LIN {X 0,Y 523.696,Z 765.358,A -85,B 0,C 180,E1 -4763.063,E2 -4763.063} C_VEL
LIN {X 0,Y 523.627,Z 770.61,A -85,B 0,C 180,E1 -4763.836,E2 -4763.836} C_VEL
LIN {X 0,Y 523.485,Z 774.989,A -85,B 0,C 180,E1 -4764.608,E2 -4764.608} C_VEL
LIN {X 0,Y 523.472,Z 780.149,A -85,B 0,C 180,E1 -4765.765,E2 -4765.765} C_VEL
LIN {X 0,Y 523.381,Z 783.938,A -85,B 0,C 180,E1 -4766.921,E2 -4766.921} C_VEL
LIN {X 0,Y 523.335,Z 785.68,A -85,B 0,C 180,E1 -4767.691,E2 -4767.691} C_VEL
LIN {X 0,Y 523.273,Z 786.929,A -85,B 0,C 180,E1 -4768.461,E2 -4768.461} C_VEL
LIN {X 0,Y 523.248,Z 787.706,A -85,B 0,C 180,E1 -4769.23,E2 -4769.23} C_VEL
LIN {X 0,Y 523.244,Z 788,A -85,B 0,C 180,E1 -4770,E2 -4770} C_VEL
LIN {X 0,Y 523.248,Z 787.707,A -85,B 0,C 180,E1 -4770.77,E2 -4770.77} C_VEL
LIN {X 0,Y 523.273,Z 786.93,A -85,B 0,C 180,E1 -4771.539,E2 -4771.539} C_VEL
LIN {X 0,Y 523.335,Z 785.682,A -85,B 0,C 180,E1 -4772.309,E2 -4772.309} C_VEL
LIN {X 0,Y 523.413,Z 782.788,A -85,B 0,C 180,E1 -4773.464,E2 -4773.464} C_VEL
LIN {X 0,Y 523.47,Z 780.149,A -85,B 0,C 180,E1 -4774.235,E2 -4774.235} C_VEL
LIN {X 0,Y 523.485,Z 774.99,A -85,B 0,C 180,E1 -4775.392,E2 -4775.392} C_VEL
LIN {X 0,Y 523.665,Z 768.76,A -85,B 0,C 180,E1 -4776.466,E2 -4776.466} C_VEL
LIN {X 0,Y 523.773,Z 760.74,A -85,B 0,C 180,E1 -4777.517,E2 -4777.517} C_VEL
LIN {X 0,Y 523.904,Z 753.36,A -85,B 0,C 180,E1 -4778.291,E2 -4778.291} C_VEL
LIN {X 0,Y 524.1,Z 745.417,A -85,B 0,C 180,E1 -4778.968,E2 -4778.968} C_VEL
LIN {X 0,Y 524.249,Z 736.974,A -85,B 0,C 180,E1 -4779.549,E2 -4779.549} C_VEL
LIN {X 0,Y 524.454,Z 726.202,A -85,B 0,C 180,E1 -4780.13,E2 -4780.13} C_VEL
LIN {X 0,Y 524.599,Z 714.549,A -85,B 0,C 180,E1 -4780.566,E2 -4780.566} C_VEL
LIN {X 0,Y 524.751,Z 704.885,A -85,B 0,C 180,E1 -4780.807,E2 -4780.807} C_VEL
LIN {X 0,Y 524.936,Z 646.273,A -85,B 0,C 180,E1 -4781.627,E2 -4781.627} C_VEL
LIN {X 0,Y 524.825,Z 633.309,A -85,B 0,C 180,E1 -4781.807,E2 -4781.807} C_VEL
LIN {X 0,Y 524.01,Z 625.533,A -85,B 0,C 180,E1 -4781.963,E2 -4781.963} C_VEL
LIN {X 0,Y 524.261,Z 604.559,A -85,B 0,C 180,E1 -4784.904,E2 -4784.904} C_VEL
LIN {X 0,Y 524.514,Z 583.003,A -85,B 0,C 180,E1 -4787.949,E2 -4787.949} C_VEL
LIN {X 0,Y 524.867,Z 561.889,A -85,B 0,C 180,E1 -4790.988,E2 -4790.988} C_VEL
LIN {X 0,Y 525.174,Z 542.146,A -85,B 0,C 180,E1 -4793.879,E2 -4793.879} C_VEL
LIN {X 0,Y 525.435,Z 522.421,A -85,B 0,C 180,E1 -4796.849,E2 -4796.849} C_VEL
LIN {X 0,Y 525.287,Z 516.932,A -85,B 0,C 180,E1 -4797.702,E2 -4797.702} C_VEL
LIN {X 0,Y 524.038,Z 510.273,A -85,B 0,C 180,E1 -4798.813,E2 -4798.813} C_VEL
LIN {X 0,Y 523.94,Z 510.034,A -85,B 0,C 180,E1 -4799.755,E2 -4799.755} C_VEL
LIN {X 0,Y 523.936,Z 510.033,A -85,B 0,C 180,E1 -4802.448,E2 -4802.448} C_VEL
LIN {X 0,Y 523.928,Z 510.036,A -85,B 0,C 180,E1 -4805.225,E2 -4805.225} C_VEL
LIN {X 0,Y 523.913,Z 510.033,A -85,B 0,C 180,E1 -4808.101,E2 -4808.101} C_VEL
LIN {X 0,Y 523.957,Z 510.03,A -85,B 0,C 180,E1 -4811.31,E2 -4811.31} C_VEL
LIN {X 0,Y 523.95,Z 510.033,A -85,B 0,C 180,E1 -4814.691,E2 -4814.691} C_VEL
LIN {X 0,Y 523.951,Z 510.025,A -85,B 0,C 180,E1 -4817.881,E2 -4817.881} C_VEL
LIN {X 0,Y 523.953,Z 510.033,A -85,B 0,C 180,E1 -4820.918,E2 -4820.918} C_VEL
LIN {X 0,Y 523.923,Z 510.029,A -85,B 0,C 180,E1 -4823.827,E2 -4823.827} C_VEL
LIN {X 0,Y 523.936,Z 510.034,A -85,B 0,C 180,E1 -4826.635,E2 -4826.635} C_VEL
LIN {X 0,Y 523.955,Z 510.029,A -85,B 0,C 180,E1 -4829.356,E2 -4829.356} C_VEL
LIN {X 0,Y 523.971,Z 510.026,A -85,B 0,C 180,E1 -4832.28,E2 -4832.28} C_VEL
LIN {X 0,Y 523.948,Z 510.03,A -85,B 0,C 180,E1 -4834.581,E2 -4834.581} C_VEL
LIN {X 0,Y 523.907,Z 510.039,A -85,B 0,C 180,E1 -4837.107,E2 -4837.107} C_VEL
LIN {X 0,Y 523.969,Z 510.024,A -85,B 0,C 180,E1 -4839.865,E2 -4839.865} C_VEL
LIN {X 0,Y 523.961,Z 510.033,A -85,B 0,C 180,E1 -4842.837,E2 -4842.837} C_VEL
LIN {X 0,Y 523.966,Z 510.03,A -85,B 0,C 180,E1 -4845.236,E2 -4845.236} C_VEL
LIN {X 0,Y 524.001,Z 510.024,A -85,B 0,C 180,E1 -4848.394,E2 -4848.394} C_VEL
LIN {X 0,Y 523.999,Z 510.023,A -85,B 0,C 180,E1 -4851.516,E2 -4851.516} C_VEL
LIN {X 0,Y 524.094,Z 510.016,A -85,B 0,C 180,E1 -4854.614,E2 -4854.614} C_VEL
LIN {X 0,Y 524.103,Z 510.01,A -85,B 0,C 180,E1 -4857.695,E2 -4857.695} C_VEL
LIN {X 0,Y 524.117,Z 510.015,A -85,B 0,C 180,E1 -4860.769,E2 -4860.769} C_VEL
LIN {X 0,Y 524.069,Z 510.019,A -85,B 0,C 180,E1 -4863.075,E2 -4863.075} C_VEL
LIN {X 0,Y 524.043,Z 510.022,A -85,B 0,C 180,E1 -4866.159,E2 -4866.159} C_VEL
LIN {X 0,Y 524.058,Z 510.143,A -85,B 0,C 180,E1 -4866.977,E2 -4866.977} C_VEL
LIN {X 0,Y 524.207,Z 511,A -85,B 0,C 180,E1 -4867.108,E2 -4867.108} C_VEL
LIN {X 0,Y 525.5,Z 515.641,A -85,B 0,C 180,E1 -4867.223,E2 -4867.223} C_VEL
LIN {X 0,Y 525.418,Z 540.428,A -85,B 0,C 180,E1 -4867.59,E2 -4867.59} C_VEL
LIN {X 0,Y 525.331,Z 553.745,A -85,B 0,C 180,E1 -4867.954,E2 -4867.954} C_VEL
LIN {X 0,Y 525.166,Z 566.276,A -85,B 0,C 180,E1 -4868.465,E2 -4868.465} C_VEL
LIN {X 0,Y 525.003,Z 577.002,A -85,B 0,C 180,E1 -4869.05,E2 -4869.05} C_VEL
LIN {X 0,Y 524.736,Z 588.282,A -85,B 0,C 180,E1 -4869.833,E2 -4869.833} C_VEL
LIN {X 0,Y 524.468,Z 598.441,A -85,B 0,C 180,E1 -4870.716,E2 -4870.716} C_VEL
LIN {X 0,Y 524.242,Z 607.233,A -85,B 0,C 180,E1 -4871.665,E2 -4871.665} C_VEL
LIN {X 0,Y 524.025,Z 615.656,A -85,B 0,C 180,E1 -4872.785,E2 -4872.785} C_VEL
LIN {X 0,Y 523.87,Z 622.807,A -85,B 0,C 180,E1 -4873.974,E2 -4873.974} C_VEL
LIN {X 0,Y 523.716,Z 628.632,A -85,B 0,C 180,E1 -4875.19,E2 -4875.19} C_VEL
LIN {X 0,Y 523.585,Z 633.022,A -85,B 0,C 180,E1 -4876.373,E2 -4876.373} C_VEL
LIN {X 0,Y 523.507,Z 636.422,A -85,B 0,C 180,E1 -4877.609,E2 -4877.609} C_VEL
LIN {X 0,Y 523.454,Z 638.654,A -85,B 0,C 180,E1 -4878.798,E2 -4878.798} C_VEL
LIN {X 0,Y 523.426,Z 639.92,A -85,B 0,C 180,E1 -4879.972,E2 -4879.972} C_VEL
LIN {X 0,Y 523.415,Z 640.261,A -85,B 0,C 180,E1 -4881.256,E2 -4881.256} C_VEL
LIN {X 0,Y 523.425,Z 639.894,A -85,B 0,C 180,E1 -4882.114,E2 -4882.114} C_VEL
LIN {X 0,Y 523.426,Z 639.12,A -85,B 0,C 180,E1 -4882.916,E2 -4882.916} C_VEL
LIN {X 0,Y 523.506,Z 637.178,A -85,B 0,C 180,E1 -4884.095,E2 -4884.095} C_VEL
LIN {X 0,Y 523.579,Z 633.768,A -85,B 0,C 180,E1 -4885.438,E2 -4885.438} C_VEL
LIN {X 0,Y 523.684,Z 629.24,A -85,B 0,C 180,E1 -4886.717,E2 -4886.717} C_VEL
LIN {X 0,Y 523.8,Z 623.233,A -85,B 0,C 180,E1 -4888.009,E2 -4888.009} C_VEL
LIN {X 0,Y 523.962,Z 616.769,A -85,B 0,C 180,E1 -4889.107,E2 -4889.107} C_VEL
LIN {X 0,Y 524.155,Z 608.949,A -85,B 0,C 180,E1 -4890.186,E2 -4890.186} C_VEL
LIN {X 0,Y 524.384,Z 600.525,A -85,B 0,C 180,E1 -4891.14,E2 -4891.14} C_VEL
LIN {X 0,Y 524.617,Z 590.534,A -85,B 0,C 180,E1 -4892.062,E2 -4892.062} C_VEL
LIN {X 0,Y 524.876,Z 580.07,A -85,B 0,C 180,E1 -4892.839,E2 -4892.839} C_VEL
LIN {X 0,Y 525.164,Z 568.003,A -85,B 0,C 180,E1 -4893.536,E2 -4893.536} C_VEL
LIN {X 0,Y 525.234,Z 562.226,A -85,B 0,C 180,E1 -4893.81,E2 -4893.81} C_VEL
LIN {X 0,Y 524.665,Z 556.768,A -85,B 0,C 180,E1 -4894.05,E2 -4894.05} C_VEL
LIN {X 0,Y 522.004,Z 547.838,A -85,B 0,C 180,E1 -4894.421,E2 -4894.421} C_VEL
LIN {X 0,Y 519.299,Z 538.713,A -85,B 0,C 180,E1 -4894.716,E2 -4894.716} C_VEL
LIN {X 0,Y 518.603,Z 532.955,A -85,B 0,C 180,E1 -4894.831,E2 -4894.831} C_VEL
LIN {X 0,Y 518.476,Z 516.07,A -85,B 0,C 180,E1 -4895.072,E2 -4895.072} C_VEL
LIN {X 0,Y 517.083,Z 511.785,A -85,B 0,C 180,E1 -4895.195,E2 -4895.195} C_VEL
LIN {X 0,Y 516.925,Z 510.992,A -85,B 0,C 180,E1 -4895.341,E2 -4895.341} C_VEL
LIN {X 0,Y 516.878,Z 510.912,A -85,B 0,C 180,E1 -4898.717,E2 -4898.717} C_VEL
LIN {X 0,Y 516.912,Z 510.907,A -85,B 0,C 180,E1 -4901.776,E2 -4901.776} C_VEL
LIN {X 0,Y 516.92,Z 510.906,A -85,B 0,C 180,E1 -4905.011,E2 -4905.011} C_VEL
LIN {X 0,Y 516.921,Z 510.902,A -85,B 0,C 180,E1 -4908.398,E2 -4908.398} C_VEL
LIN {X 0,Y 516.885,Z 510.914,A -85,B 0,C 180,E1 -4911.286,E2 -4911.286} C_VEL
LIN {X 0,Y 516.87,Z 510.909,A -85,B 0,C 180,E1 -4914.221,E2 -4914.221} C_VEL
LIN {X 0,Y 516.896,Z 510.908,A -85,B 0,C 180,E1 -4917.054,E2 -4917.054} C_VEL
LIN {X 0,Y 516.893,Z 510.91,A -85,B 0,C 180,E1 -4919.797,E2 -4919.797} C_VEL
LIN {X 0,Y 516.931,Z 510.901,A -85,B 0,C 180,E1 -4922.468,E2 -4922.468} C_VEL
LIN {X 0,Y 516.911,Z 510.906,A -85,B 0,C 180,E1 -4925.073,E2 -4925.073} C_VEL
LIN {X 0,Y 516.888,Z 510.906,A -85,B 0,C 180,E1 -4928.463,E2 -4928.463} C_VEL
LIN {X 0,Y 516.903,Z 510.905,A -85,B 0,C 180,E1 -4930.955,E2 -4930.955} C_VEL
LIN {X 0,Y 516.91,Z 510.91,A -85,B 0,C 180,E1 -4933.411,E2 -4933.411} C_VEL
LIN {X 0,Y 516.899,Z 510.911,A -85,B 0,C 180,E1 -4935.834,E2 -4935.834} C_VEL
LIN {X 0,Y 516.971,Z 510.897,A -85,B 0,C 180,E1 -4938.234,E2 -4938.234} C_VEL
LIN {X 0,Y 516.97,Z 510.901,A -85,B 0,C 180,E1 -4941.4,E2 -4941.4} C_VEL
LIN {X 0,Y 517.026,Z 510.889,A -85,B 0,C 180,E1 -4944.54,E2 -4944.54} C_VEL
LIN {X 0,Y 517.088,Z 510.89,A -85,B 0,C 180,E1 -4947.663,E2 -4947.663} C_VEL
LIN {X 0,Y 517.097,Z 510.88,A -85,B 0,C 180,E1 -4950.779,E2 -4950.779} C_VEL
LIN {X 0,Y 517.016,Z 510.891,A -85,B 0,C 180,E1 -4953.117,E2 -4953.117} C_VEL
LIN {X 0,Y 516.993,Z 510.896,A -85,B 0,C 180,E1 -4956.243,E2 -4956.243} C_VEL
LIN {X 0,Y 516.954,Z 510.901,A -85,B 0,C 180,E1 -4959.389,E2 -4959.389} C_VEL
LIN {X 0,Y 516.958,Z 510.907,A -85,B 0,C 180,E1 -4961.807,E2 -4961.807} C_VEL
LIN {X 0,Y 516.949,Z 510.899,A -85,B 0,C 180,E1 -4965.146,E2 -4965.146} C_VEL
LIN {X 0,Y 516.929,Z 510.905,A -85,B 0,C 180,E1 -4968.222,E2 -4968.222} C_VEL
LIN {X 0,Y 516.916,Z 510.903,A -85,B 0,C 180,E1 -4970.701,E2 -4970.701} C_VEL
LIN {X 0,Y 516.894,Z 510.913,A -85,B 0,C 180,E1 -4974.072,E2 -4974.072} C_VEL
LIN {X 0,Y 516.928,Z 510.902,A -85,B 0,C 180,E1 -4976.657,E2 -4976.657} C_VEL
LIN {X 0,Y 516.913,Z 510.906,A -85,B 0,C 180,E1 -4979.523,E2 -4979.523} C_VEL
LIN {X 0,Y 516.896,Z 510.907,A -85,B 0,C 180,E1 -4982.543,E2 -4982.543} C_VEL
LIN {X 0,Y 516.866,Z 510.91,A -85,B 0,C 180,E1 -4985.329,E2 -4985.329} C_VEL
LIN {X 0,Y 516.881,Z 510.915,A -85,B 0,C 180,E1 -4987.942,E2 -4987.942} C_VEL
LIN {X 0,Y 516.903,Z 510.905,A -85,B 0,C 180,E1 -4990.739,E2 -4990.739} C_VEL
LIN {X 0,Y 516.881,Z 510.913,A -85,B 0,C 180,E1 -4993.902,E2 -4993.902} C_VEL
LIN {X 0,Y 516.88,Z 510.917,A -85,B 0,C 180,E1 -4996.106,E2 -4996.106} C_VEL
LIN {X 0,Y 516.914,Z 510.908,A -85,B 0,C 180,E1 -4998.397,E2 -4998.397} C_VEL
LIN {X 0,Y 516.879,Z 510.907,A -85,B 0,C 180,E1 -5001.283,E2 -5001.283} C_VEL
LIN {X 0,Y 516.886,Z 510.916,A -85,B 0,C 180,E1 -5004.22,E2 -5004.22} C_VEL
LIN {X 0,Y 516.893,Z 510.906,A -85,B 0,C 180,E1 -5007.052,E2 -5007.052} C_VEL
LIN {X 0,Y 516.897,Z 510.908,A -85,B 0,C 180,E1 -5009.796,E2 -5009.796} C_VEL
LIN {X 0,Y 516.924,Z 510.908,A -85,B 0,C 180,E1 -5012.467,E2 -5012.467} C_VEL
LIN {X 0,Y 516.905,Z 510.904,A -85,B 0,C 180,E1 -5015.071,E2 -5015.071} C_VEL
LIN {X 0,Y 516.88,Z 510.914,A -85,B 0,C 180,E1 -5018.462,E2 -5018.462} C_VEL
LIN {X 0,Y 516.897,Z 510.906,A -85,B 0,C 180,E1 -5020.954,E2 -5020.954} C_VEL
LIN {X 0,Y 516.909,Z 510.903,A -85,B 0,C 180,E1 -5023.41,E2 -5023.41} C_VEL
LIN {X 0,Y 516.887,Z 510.908,A -85,B 0,C 180,E1 -5025.833,E2 -5025.833} C_VEL
LIN {X 0,Y 516.996,Z 510.9,A -85,B 0,C 180,E1 -5028.234,E2 -5028.234} C_VEL
LIN {X 0,Y 516.963,Z 510.897,A -85,B 0,C 180,E1 -5031.399,E2 -5031.399} C_VEL
LIN {X 0,Y 517.051,Z 510.894,A -85,B 0,C 180,E1 -5034.54,E2 -5034.54} C_VEL
LIN {X 0,Y 517.076,Z 510.883,A -85,B 0,C 180,E1 -5037.663,E2 -5037.663} C_VEL
LIN {X 0,Y 517.086,Z 510.886,A -85,B 0,C 180,E1 -5040.778,E2 -5040.778} C_VEL
LIN {X 0,Y 517.008,Z 510.893,A -85,B 0,C 180,E1 -5043.117,E2 -5043.117} C_VEL
LIN {X 0,Y 517.001,Z 510.897,A -85,B 0,C 180,E1 -5046.243,E2 -5046.243} C_VEL
LIN {X 0,Y 516.947,Z 510.899,A -85,B 0,C 180,E1 -5049.389,E2 -5049.389} C_VEL
LIN {X 0,Y 516.942,Z 510.9,A -85,B 0,C 180,E1 -5051.807,E2 -5051.807} C_VEL
LIN {X 0,Y 516.937,Z 510.902,A -85,B 0,C 180,E1 -5055.148,E2 -5055.148} C_VEL
LIN {X 0,Y 516.917,Z 510.906,A -85,B 0,C 180,E1 -5058.222,E2 -5058.222} C_VEL
LIN {X 0,Y 516.904,Z 510.913,A -85,B 0,C 180,E1 -5060.702,E2 -5060.702} C_VEL
LIN {X 0,Y 516.902,Z 510.906,A -85,B 0,C 180,E1 -5064.072,E2 -5064.072} C_VEL
LIN {X 0,Y 516.921,Z 510.911,A -85,B 0,C 180,E1 -5066.658,E2 -5066.658} C_VEL
LIN {X 0,Y 516.917,Z 510.903,A -85,B 0,C 180,E1 -5069.527,E2 -5069.527} C_VEL
LIN {X 0,Y 516.893,Z 510.912,A -85,B 0,C 180,E1 -5072.545,E2 -5072.545} C_VEL
LIN {X 0,Y 516.877,Z 510.909,A -85,B 0,C 180,E1 -5075.333,E2 -5075.333} C_VEL
LIN {X 0,Y 516.875,Z 510.908,A -85,B 0,C 180,E1 -5077.944,E2 -5077.944} C_VEL
LIN {X 0,Y 516.879,Z 510.916,A -85,B 0,C 180,E1 -5080.742,E2 -5080.742} C_VEL
LIN {X 0,Y 516.897,Z 510.915,A -85,B 0,C 180,E1 -5082.83,E2 -5082.83} C_VEL
LIN {X 0,Y 516.917,Z 510.91,A -85,B 0,C 180,E1 -5085.011,E2 -5085.011} C_VEL
LIN {X 0,Y 516.913,Z 510.906,A -85,B 0,C 180,E1 -5088.399,E2 -5088.399} C_VEL
LIN {X 0,Y 516.879,Z 510.911,A -85,B 0,C 180,E1 -5091.285,E2 -5091.285} C_VEL
LIN {X 0,Y 516.884,Z 510.909,A -85,B 0,C 180,E1 -5094.222,E2 -5094.222} C_VEL
LIN {X 0,Y 516.895,Z 510.914,A -85,B 0,C 180,E1 -5097.054,E2 -5097.054} C_VEL
LIN {X 0,Y 516.932,Z 511.029,A -85,B 0,C 180,E1 -5100.366,E2 -5100.366} C_VEL
LIN {X 0,Y 518.923,Z 520.98,A -85,B 0,C 180,E1 -5102.145,E2 -5102.145} C_VEL
LIN {X 0,Y 518.947,Z 529.197,A -85,B 0,C 180,E1 -5103.455,E2 -5103.455} C_VEL
LIN {X 0,Y 518.414,Z 548.211,A -85,B 0,C 180,E1 -5106.427,E2 -5106.427} C_VEL
LIN {X 0,Y 517.913,Z 567.608,A -85,B 0,C 180,E1 -5109.442,E2 -5109.442} C_VEL
LIN {X 0,Y 517.521,Z 584.748,A -85,B 0,C 180,E1 -5112.019,E2 -5112.019} C_VEL
LIN {X 0,Y 517.208,Z 606.759,A -85,B 0,C 180,E1 -5115.24,E2 -5115.24} C_VEL
LIN {X 0,Y 516.951,Z 624.671,A -85,B 0,C 180,E1 -5117.852,E2 -5117.852} C_VEL
LIN {X 0,Y 518.066,Z 636.508,A -85,B 0,C 180,E1 -5118.065,E2 -5118.065} C_VEL
LIN {X 0,Y 517.848,Z 703.106,A -85,B 0,C 180,E1 -5119.023,E2 -5119.023} C_VEL
LIN {X 0,Y 517.6,Z 713.015,A -85,B 0,C 180,E1 -5119.265,E2 -5119.265} C_VEL
LIN {X 0,Y 517.507,Z 724.237,A -85,B 0,C 180,E1 -5119.683,E2 -5119.683} C_VEL
LIN {X 0,Y 517.255,Z 734.516,A -85,B 0,C 180,E1 -5120.222,E2 -5120.222} C_VEL
LIN {X 0,Y 517.086,Z 744.454,A -85,B 0,C 180,E1 -5120.909,E2 -5120.909} C_VEL
LIN {X 0,Y 516.857,Z 752.427,A -85,B 0,C 180,E1 -5121.595,E2 -5121.595} C_VEL
LIN {X 0,Y 516.704,Z 759.897,A -85,B 0,C 180,E1 -5122.379,E2 -5122.379} C_VEL
LIN {X 0,Y 516.591,Z 766.92,A -85,B 0,C 180,E1 -5123.281,E2 -5123.281} C_VEL
LIN {X 0,Y 516.496,Z 773.47,A -85,B 0,C 180,E1 -5124.339,E2 -5124.339} C_VEL
LIN {X 0,Y 516.322,Z 778.169,A -85,B 0,C 180,E1 -5125.315,E2 -5125.315} C_VEL
LIN {X 0,Y 516.385,Z 781.242,A -85,B 0,C 180,E1 -5126.098,E2 -5126.098} C_VEL
LIN {X 0,Y 516.295,Z 783.609,A -85,B 0,C 180,E1 -5126.879,E2 -5126.879} C_VEL
LIN {X 0,Y 516.262,Z 785.398,A -85,B 0,C 180,E1 -5127.659,E2 -5127.659} C_VEL
LIN {X 0,Y 516.19,Z 786.673,A -85,B 0,C 180,E1 -5128.44,E2 -5128.44} C_VEL
LIN {X 0,Y 516.158,Z 787.467,A -85,B 0,C 180,E1 -5129.22,E2 -5129.22} C_VEL
LIN {X 0,Y 516.151,Z 787.768,A -85,B 0,C 180,E1 -5130,E2 -5130} C_VEL
LIN {X 0,Y 516.158,Z 787.469,A -85,B 0,C 180,E1 -5130.78,E2 -5130.78} C_VEL
LIN {X 0,Y 516.19,Z 786.674,A -85,B 0,C 180,E1 -5131.56,E2 -5131.56} C_VEL
LIN {X 0,Y 516.262,Z 785.398,A -85,B 0,C 180,E1 -5132.34,E2 -5132.34} C_VEL
LIN {X 0,Y 516.33,Z 782.429,A -85,B 0,C 180,E1 -5133.512,E2 -5133.512} C_VEL
LIN {X 0,Y 516.376,Z 779.716,A -85,B 0,C 180,E1 -5134.293,E2 -5134.293} C_VEL
LIN {X 0,Y 516.432,Z 774.416,A -85,B 0,C 180,E1 -5135.466,E2 -5135.466} C_VEL
LIN {X 0,Y 516.565,Z 768.545,A -85,B 0,C 180,E1 -5136.474,E2 -5136.474} C_VEL
LIN {X 0,Y 516.672,Z 761.524,A -85,B 0,C 180,E1 -5137.424,E2 -5137.424} C_VEL
LIN {X 0,Y 516.814,Z 753.324,A -85,B 0,C 180,E1 -5138.307,E2 -5138.307} C_VEL
LIN {X 0,Y 517.014,Z 745.516,A -85,B 0,C 180,E1 -5138.993,E2 -5138.993} C_VEL
LIN {X 0,Y 517.183,Z 737.327,A -85,B 0,C 180,E1 -5139.582,E2 -5139.582} C_VEL
LIN {X 0,Y 517.322,Z 728.859,A -85,B 0,C 180,E1 -5140.073,E2 -5140.073} C_VEL
LIN {X 0,Y 517.556,Z 719.044,A -85,B 0,C 180,E1 -5140.513,E2 -5140.513} C_VEL
LIN {X 0,Y 517.709,Z 707.406,A -85,B 0,C 180,E1 -5140.881,E2 -5140.881} C_VEL
LIN {X 0,Y 517.853,Z 689.806,A -85,B 0,C 180,E1 -5141.175,E2 -5141.175} C_VEL
LIN {X 0,Y 517.893,Z 634.084,A -85,B 0,C 180,E1 -5141.948,E2 -5141.948} C_VEL
LIN {X 0,Y 516.928,Z 624.065,A -85,B 0,C 180,E1 -5142.141,E2 -5142.141} C_VEL
LIN {X 0,Y 517.185,Z 605.597,A -85,B 0,C 180,E1 -5144.761,E2 -5144.761} C_VEL
LIN {X 0,Y 517.441,Z 583.365,A -85,B 0,C 180,E1 -5147.962,E2 -5147.962} C_VEL
LIN {X 0,Y 517.767,Z 563.429,A -85,B 0,C 180,E1 -5150.873,E2 -5150.873} C_VEL
LIN {X 0,Y 518.073,Z 545.172,A -85,B 0,C 180,E1 -5153.589,E2 -5153.589} C_VEL
LIN {X 0,Y 518.443,Z 525.628,A -85,B 0,C 180,E1 -5156.573,E2 -5156.573} C_VEL
LIN {X 0,Y 518.407,Z 518.846,A -85,B 0,C 180,E1 -5157.639,E2 -5157.639} C_VEL
LIN {X 0,Y 516.969,Z 511.076,A -85,B 0,C 180,E1 -5158.966,E2 -5158.966} C_VEL
LIN {X 0,Y 516.879,Z 510.91,A -85,B 0,C 180,E1 -5162.024,E2 -5162.024} C_VEL
LIN {X 0,Y 516.888,Z 510.915,A -85,B 0,C 180,E1 -5164.823,E2 -5164.823} C_VEL
LIN {X 0,Y 516.877,Z 510.909,A -85,B 0,C 180,E1 -5167.943,E2 -5167.943} C_VEL
LIN {X 0,Y 516.881,Z 510.914,A -85,B 0,C 180,E1 -5170.741,E2 -5170.741} C_VEL
LIN {X 0,Y 516.9,Z 510.912,A -85,B 0,C 180,E1 -5172.828,E2 -5172.828} C_VEL
LIN {X 0,Y 516.916,Z 510.91,A -85,B 0,C 180,E1 -5175.009,E2 -5175.009} C_VEL
LIN {X 0,Y 516.916,Z 510.903,A -85,B 0,C 180,E1 -5178.397,E2 -5178.397} C_VEL
LIN {X 0,Y 516.9,Z 510.909,A -85,B 0,C 180,E1 -5181.286,E2 -5181.286} C_VEL
LIN {X 0,Y 516.885,Z 510.907,A -85,B 0,C 180,E1 -5184.221,E2 -5184.221} C_VEL
LIN {X 0,Y 516.89,Z 510.912,A -85,B 0,C 180,E1 -5187.053,E2 -5187.053} C_VEL
LIN {X 0,Y 516.893,Z 510.906,A -85,B 0,C 180,E1 -5189.797,E2 -5189.797} C_VEL
LIN {X 0,Y 516.922,Z 510.906,A -85,B 0,C 180,E1 -5192.467,E2 -5192.467} C_VEL
LIN {X 0,Y 516.904,Z 510.912,A -85,B 0,C 180,E1 -5195.072,E2 -5195.072} C_VEL
LIN {X 0,Y 516.877,Z 510.912,A -85,B 0,C 180,E1 -5198.462,E2 -5198.462} C_VEL
LIN {X 0,Y 516.898,Z 510.914,A -85,B 0,C 180,E1 -5200.955,E2 -5200.955} C_VEL
LIN {X 0,Y 516.908,Z 510.907,A -85,B 0,C 180,E1 -5203.41,E2 -5203.41} C_VEL
LIN {X 0,Y 516.886,Z 510.908,A -85,B 0,C 180,E1 -5205.834,E2 -5205.834} C_VEL
LIN {X 0,Y 516.994,Z 510.896,A -85,B 0,C 180,E1 -5208.235,E2 -5208.235} C_VEL
LIN {X 0,Y 516.963,Z 510.901,A -85,B 0,C 180,E1 -5211.4,E2 -5211.4} C_VEL
LIN {X 0,Y 517.054,Z 510.892,A -85,B 0,C 180,E1 -5214.541,E2 -5214.541} C_VEL
LIN {X 0,Y 517.076,Z 510.885,A -85,B 0,C 180,E1 -5217.663,E2 -5217.663} C_VEL
LIN {X 0,Y 517.087,Z 510.891,A -85,B 0,C 180,E1 -5220.779,E2 -5220.779} C_VEL
LIN {X 0,Y 517.01,Z 510.898,A -85,B 0,C 180,E1 -5223.117,E2 -5223.117} C_VEL
LIN {X 0,Y 517.006,Z 510.899,A -85,B 0,C 180,E1 -5226.244,E2 -5226.244} C_VEL
LIN {X 0,Y 517.026,Z 511.162,A -85,B 0,C 180,E1 -5226.851,E2 -5226.851} C_VEL
LIN {X 0,Y 517.282,Z 512.234,A -85,B 0,C 180,E1 -5226.961,E2 -5226.961} C_VEL
LIN {X 0,Y 518.586,Z 517.279,A -85,B 0,C 180,E1 -5227.073,E2 -5227.073} C_VEL
LIN {X 0,Y 518.491,Z 541.4,A -85,B 0,C 180,E1 -5227.434,E2 -5227.434} C_VEL
LIN {X 0,Y 518.415,Z 554.495,A -85,B 0,C 180,E1 -5227.792,E2 -5227.792} C_VEL
LIN {X 0,Y 518.272,Z 566.108,A -85,B 0,C 180,E1 -5228.257,E2 -5228.257} C_VEL
LIN {X 0,Y 518.113,Z 577.551,A -85,B 0,C 180,E1 -5228.876,E2 -5228.876} C_VEL
LIN {X 0,Y 517.844,Z 588.947,A -85,B 0,C 180,E1 -5229.669,E2 -5229.669} C_VEL
LIN {X 0,Y 517.55,Z 599.194,A -85,B 0,C 180,E1 -5230.564,E2 -5230.564} C_VEL
LIN {X 0,Y 517.292,Z 608.336,A -85,B 0,C 180,E1 -5231.56,E2 -5231.56} C_VEL
LIN {X 0,Y 517.053,Z 617.197,A -85,B 0,C 180,E1 -5232.761,E2 -5232.761} C_VEL
LIN {X 0,Y 516.895,Z 624.271,A -85,B 0,C 180,E1 -5233.966,E2 -5233.966} C_VEL
LIN {X 0,Y 516.704,Z 630.546,A -85,B 0,C 180,E1 -5235.341,E2 -5235.341} C_VEL
LIN {X 0,Y 516.579,Z 634.913,A -85,B 0,C 180,E1 -5236.601,E2 -5236.601} C_VEL
LIN {X 0,Y 516.505,Z 637.81,A -85,B 0,C 180,E1 -5237.739,E2 -5237.739} C_VEL
LIN {X 0,Y 516.436,Z 640.064,A -85,B 0,C 180,E1 -5239.063,E2 -5239.063} C_VEL
LIN {X 0,Y 516.408,Z 641.014,A -85,B 0,C 180,E1 -5240.112,E2 -5240.112} C_VEL
LIN {X 0,Y 516.381,Z 641.197,A -85,B 0,C 180,E1 -5241.56,E2 -5241.56} C_VEL
LIN {X 0,Y 516.414,Z 640.678,A -85,B 0,C 180,E1 -5242.4,E2 -5242.4} C_VEL
LIN {X 0,Y 516.438,Z 639.688,A -85,B 0,C 180,E1 -5243.244,E2 -5243.244} C_VEL
LIN {X 0,Y 516.485,Z 637.892,A -85,B 0,C 180,E1 -5244.263,E2 -5244.263} C_VEL
LIN {X 0,Y 516.587,Z 633.766,A -85,B 0,C 180,E1 -5245.808,E2 -5245.808} C_VEL
LIN {X 0,Y 516.739,Z 628.884,A -85,B 0,C 180,E1 -5247.105,E2 -5247.105} C_VEL
LIN {X 0,Y 516.866,Z 622.439,A -85,B 0,C 180,E1 -5248.419,E2 -5248.419} C_VEL
LIN {X 0,Y 517.084,Z 615.358,A -85,B 0,C 180,E1 -5249.56,E2 -5249.56} C_VEL
LIN {X 0,Y 517.286,Z 607.222,A -85,B 0,C 180,E1 -5250.63,E2 -5250.63} C_VEL
LIN {X 0,Y 517.55,Z 597.771,A -85,B 0,C 180,E1 -5251.635,E2 -5251.635} C_VEL
LIN {X 0,Y 517.825,Z 587.493,A -85,B 0,C 180,E1 -5252.515,E2 -5252.515} C_VEL
LIN {X 0,Y 518.054,Z 577.412,A -85,B 0,C 180,E1 -5253.212,E2 -5253.212} C_VEL
LIN {X 0,Y 518.283,Z 565.658,A -85,B 0,C 180,E1 -5253.853,E2 -5253.853} C_VEL
LIN {X 0,Y 518.444,Z 552.926,A -85,B 0,C 180,E1 -5254.361,E2 -5254.361} C_VEL
LIN {X 0,Y 518.563,Z 539.177,A -85,B 0,C 180,E1 -5254.726,E2 -5254.726} C_VEL
LIN {X 0,Y 518.603,Z 532.955,A -85,B 0,C 180,E1 -5254.831,E2 -5254.831} C_VEL
LIN {X 0,Y 517.998,Z 529.111,A -85,B 0,C 180,E1 -5254.902,E2 -5254.902} C_VEL
LIN {X 0,Y 515.377,Z 523.171,A -85,B 0,C 180,E1 -5255.054,E2 -5255.054} C_VEL
LIN {X 0,Y 511.457,Z 516.232,A -85,B 0,C 180,E1 -5255.258,E2 -5255.258} C_VEL
LIN {X 0,Y 510.401,Z 513.803,A -85,B 0,C 180,E1 -5255.324,E2 -5255.324} C_VEL
LIN {X 0,Y 509.963,Z 512.303,A -85,B 0,C 180,E1 -5255.412,E2 -5255.412} C_VEL
LIN {X 0,Y 509.871,Z 511.819,A -85,B 0,C 180,E1 -5255.587,E2 -5255.587} C_VEL
LIN {X 0,Y 509.846,Z 511.787,A -85,B 0,C 180,E1 -5258.339,E2 -5258.339} C_VEL
LIN {X 0,Y 509.855,Z 511.792,A -85,B 0,C 180,E1 -5261.426,E2 -5261.426} C_VEL
LIN {X 0,Y 509.854,Z 511.783,A -85,B 0,C 180,E1 -5264.669,E2 -5264.669} C_VEL
LIN {X 0,Y 509.862,Z 511.782,A -85,B 0,C 180,E1 -5268.103,E2 -5268.103} C_VEL
LIN {X 0,Y 509.859,Z 511.782,A -85,B 0,C 180,E1 -5270.65,E2 -5270.65} C_VEL
LIN {X 0,Y 509.824,Z 511.792,A -85,B 0,C 180,E1 -5273.648,E2 -5273.648} C_VEL
LIN {X 0,Y 509.859,Z 511.782,A -85,B 0,C 180,E1 -5276.54,E2 -5276.54} C_VEL
LIN {X 0,Y 509.846,Z 511.79,A -85,B 0,C 180,E1 -5279.335,E2 -5279.335} C_VEL
LIN {X 0,Y 509.896,Z 511.779,A -85,B 0,C 180,E1 -5282.055,E2 -5282.055} C_VEL
LIN {X 0,Y 509.878,Z 511.78,A -85,B 0,C 180,E1 -5284.705,E2 -5284.705} C_VEL
LIN {X 0,Y 509.829,Z 511.793,A -85,B 0,C 180,E1 -5287.459,E2 -5287.459} C_VEL
LIN {X 0,Y 509.92,Z 511.779,A -85,B 0,C 180,E1 -5289.845,E2 -5289.845} C_VEL
LIN {X 0,Y 509.877,Z 511.783,A -85,B 0,C 180,E1 -5293.175,E2 -5293.175} C_VEL
LIN {X 0,Y 509.868,Z 511.79,A -85,B 0,C 180,E1 -5295.635,E2 -5295.635} C_VEL
LIN {X 0,Y 509.917,Z 511.775,A -85,B 0,C 180,E1 -5298.875,E2 -5298.875} C_VEL
LIN {X 0,Y 509.956,Z 511.773,A -85,B 0,C 180,E1 -5302.079,E2 -5302.079} C_VEL
LIN {X 0,Y 509.977,Z 511.767,A -85,B 0,C 180,E1 -5304.464,E2 -5304.464} C_VEL
LIN {X 0,Y 510.059,Z 511.765,A -85,B 0,C 180,E1 -5307.631,E2 -5307.631} C_VEL
LIN {X 0,Y 510.068,Z 511.756,A -85,B 0,C 180,E1 -5310.79,E2 -5310.79} C_VEL
LIN {X 0,Y 509.958,Z 511.771,A -85,B 0,C 180,E1 -5313.16,E2 -5313.16} C_VEL
LIN {X 0,Y 509.941,Z 511.773,A -85,B 0,C 180,E1 -5316.33,E2 -5316.33} C_VEL
LIN {X 0,Y 509.912,Z 511.775,A -85,B 0,C 180,E1 -5318.72,E2 -5318.72} C_VEL
LIN {X 0,Y 509.909,Z 511.783,A -85,B 0,C 180,E1 -5321.931,E2 -5321.931} C_VEL
LIN {X 0,Y 509.899,Z 511.778,A -85,B 0,C 180,E1 -5325.241,E2 -5325.241} C_VEL
LIN {X 0,Y 509.893,Z 511.785,A -85,B 0,C 180,E1 -5328,E2 -5328} C_VEL
LIN {X 0,Y 509.854,Z 511.782,A -85,B 0,C 180,E1 -5331.001,E2 -5331.001} C_VEL
LIN {X 0,Y 509.825,Z 511.79,A -85,B 0,C 180,E1 -5333.563,E2 -5333.563} C_VEL
LIN {X 0,Y 509.914,Z 511.778,A -85,B 0,C 180,E1 -5336.378,E2 -5336.378} C_VEL
LIN {X 0,Y 509.878,Z 511.779,A -85,B 0,C 180,E1 -5338.843,E2 -5338.843} C_VEL
LIN {X 0,Y 509.821,Z 511.79,A -85,B 0,C 180,E1 -5341.589,E2 -5341.589} C_VEL
LIN {X 0,Y 509.847,Z 511.787,A -85,B 0,C 180,E1 -5344.413,E2 -5344.413} C_VEL
LIN {X 0,Y 509.817,Z 511.788,A -85,B 0,C 180,E1 -5347.34,E2 -5347.34} C_VEL
LIN {X 0,Y 509.861,Z 511.786,A -85,B 0,C 180,E1 -5350.379,E2 -5350.379} C_VEL
LIN {X 0,Y 509.838,Z 511.784,A -85,B 0,C 180,E1 -5353.063,E2 -5353.063} C_VEL
LIN {X 0,Y 509.828,Z 511.79,A -85,B 0,C 180,E1 -5355.791,E2 -5355.791} C_VEL
LIN {X 0,Y 509.855,Z 511.785,A -85,B 0,C 180,E1 -5358.574,E2 -5358.574} C_VEL
LIN {X 0,Y 509.848,Z 511.787,A -85,B 0,C 180,E1 -5361.785,E2 -5361.785} C_VEL
LIN {X 0,Y 509.842,Z 511.787,A -85,B 0,C 180,E1 -5364.622,E2 -5364.622} C_VEL
LIN {X 0,Y 509.861,Z 511.782,A -85,B 0,C 180,E1 -5367.48,E2 -5367.48} C_VEL
LIN {X 0,Y 509.876,Z 511.789,A -85,B 0,C 180,E1 -5370.268,E2 -5370.268} C_VEL
LIN {X 0,Y 509.881,Z 511.78,A -85,B 0,C 180,E1 -5372.944,E2 -5372.944} C_VEL
LIN {X 0,Y 509.863,Z 511.782,A -85,B 0,C 180,E1 -5375.573,E2 -5375.573} C_VEL
LIN {X 0,Y 509.844,Z 511.784,A -85,B 0,C 180,E1 -5378.998,E2 -5378.998} C_VEL
LIN {X 0,Y 509.881,Z 511.783,A -85,B 0,C 180,E1 -5381.998,E2 -5381.998} C_VEL
LIN {X 0,Y 509.902,Z 511.779,A -85,B 0,C 180,E1 -5384.818,E2 -5384.818} C_VEL
LIN {X 0,Y 509.935,Z 511.777,A -85,B 0,C 180,E1 -5388.1,E2 -5388.1} C_VEL
LIN {X 0,Y 509.91,Z 511.775,A -85,B 0,C 180,E1 -5391.279,E2 -5391.279} C_VEL
LIN {X 0,Y 509.97,Z 511.768,A -85,B 0,C 180,E1 -5393.67,E2 -5393.67} C_VEL
LIN {X 0,Y 509.95,Z 511.774,A -85,B 0,C 180,E1 -5396.84,E2 -5396.84} C_VEL
LIN {X 0,Y 510.056,Z 511.758,A -85,B 0,C 180,E1 -5399.21,E2 -5399.21} C_VEL
LIN {X 0,Y 510.046,Z 511.766,A -85,B 0,C 180,E1 -5402.369,E2 -5402.369} C_VEL
LIN {X 0,Y 509.969,Z 511.774,A -85,B 0,C 180,E1 -5406.329,E2 -5406.329} C_VEL
LIN {X 0,Y 509.909,Z 511.782,A -85,B 0,C 180,E1 -5408.72,E2 -5408.72} C_VEL
LIN {X 0,Y 509.894,Z 511.778,A -85,B 0,C 180,E1 -5411.932,E2 -5411.932} C_VEL
LIN {X 0,Y 509.884,Z 511.78,A -85,B 0,C 180,E1 -5415.242,E2 -5415.242} C_VEL
LIN {X 0,Y 509.879,Z 511.78,A -85,B 0,C 180,E1 -5418.001,E2 -5418.001} C_VEL
LIN {X 0,Y 509.842,Z 511.788,A -85,B 0,C 180,E1 -5421.002,E2 -5421.002} C_VEL
LIN {X 0,Y 509.828,Z 511.786,A -85,B 0,C 180,E1 -5423.563,E2 -5423.563} C_VEL
LIN {X 0,Y 509.905,Z 511.78,A -85,B 0,C 180,E1 -5426.379,E2 -5426.379} C_VEL
LIN {X 0,Y 509.878,Z 511.787,A -85,B 0,C 180,E1 -5428.844,E2 -5428.844} C_VEL
LIN {X 0,Y 509.818,Z 511.787,A -85,B 0,C 180,E1 -5431.59,E2 -5431.59} C_VEL
LIN {X 0,Y 509.848,Z 511.787,A -85,B 0,C 180,E1 -5434.414,E2 -5434.414} C_VEL
LIN {X 0,Y 509.812,Z 511.789,A -85,B 0,C 180,E1 -5437.341,E2 -5437.341} C_VEL
LIN {X 0,Y 509.832,Z 511.788,A -85,B 0,C 180,E1 -5440.383,E2 -5440.383} C_VEL
LIN {X 0,Y 509.832,Z 511.791,A -85,B 0,C 180,E1 -5443.065,E2 -5443.065} C_VEL
LIN {X 0,Y 509.825,Z 511.786,A -85,B 0,C 180,E1 -5445.793,E2 -5445.793} C_VEL
LIN {X 0,Y 509.854,Z 511.787,A -85,B 0,C 180,E1 -5448.575,E2 -5448.575} C_VEL
LIN {X 0,Y 509.848,Z 511.783,A -85,B 0,C 180,E1 -5451.787,E2 -5451.787} C_VEL
LIN {X 0,Y 509.839,Z 511.79,A -85,B 0,C 180,E1 -5454.624,E2 -5454.624} C_VEL
LIN {X 0,Y 509.863,Z 511.788,A -85,B 0,C 180,E1 -5457.482,E2 -5457.482} C_VEL
LIN {X 0,Y 509.912,Z 511.99,A -85,B 0,C 180,E1 -5460.196,E2 -5460.196} C_VEL
LIN {X 0,Y 512.075,Z 523.14,A -85,B 0,C 180,E1 -5462.185,E2 -5462.185} C_VEL
LIN {X 0,Y 511.878,Z 533.986,A -85,B 0,C 180,E1 -5463.938,E2 -5463.938} C_VEL
LIN {X 0,Y 511.351,Z 552.4,A -85,B 0,C 180,E1 -5466.869,E2 -5466.869} C_VEL
LIN {X 0,Y 510.773,Z 572.895,A -85,B 0,C 180,E1 -5470.09,E2 -5470.09} C_VEL
LIN {X 0,Y 510.437,Z 589.341,A -85,B 0,C 180,E1 -5472.575,E2 -5472.575} C_VEL
LIN {X 0,Y 510.096,Z 610.033,A -85,B 0,C 180,E1 -5475.641,E2 -5475.641} C_VEL
LIN {X 0,Y 509.882,Z 623.464,A -85,B 0,C 180,E1 -5477.654,E2 -5477.654} C_VEL
LIN {X 0,Y 510.954,Z 634.279,A -85,B 0,C 180,E1 -5477.86,E2 -5477.86} C_VEL
LIN {X 0,Y 510.979,Z 665.653,A -85,B 0,C 180,E1 -5478.32,E2 -5478.32} C_VEL
LIN {X 0,Y 510.831,Z 703.726,A -85,B 0,C 180,E1 -5478.895,E2 -5478.895} C_VEL
LIN {X 0,Y 510.598,Z 716.003,A -85,B 0,C 180,E1 -5479.241,E2 -5479.241} C_VEL
LIN {X 0,Y 510.38,Z 726.331,A -85,B 0,C 180,E1 -5479.688,E2 -5479.688} C_VEL
LIN {X 0,Y 510.179,Z 735.081,A -85,B 0,C 180,E1 -5480.185,E2 -5480.185} C_VEL
LIN {X 0,Y 510.001,Z 744.733,A -85,B 0,C 180,E1 -5480.882,E2 -5480.882} C_VEL
LIN {X 0,Y 509.725,Z 753.52,A -85,B 0,C 180,E1 -5481.676,E2 -5481.676} C_VEL
LIN {X 0,Y 509.562,Z 762.185,A -85,B 0,C 180,E1 -5482.67,E2 -5482.67} C_VEL
LIN {X 0,Y 509.457,Z 769,A -85,B 0,C 180,E1 -5483.664,E2 -5483.664} C_VEL
LIN {X 0,Y 509.382,Z 773.479,A -85,B 0,C 180,E1 -5484.458,E2 -5484.458} C_VEL
LIN {X 0,Y 509.304,Z 778.763,A -85,B 0,C 180,E1 -5485.647,E2 -5485.647} C_VEL
LIN {X 0,Y 509.279,Z 781.469,A -85,B 0,C 180,E1 -5486.44,E2 -5486.44} C_VEL
LIN {X 0,Y 509.214,Z 784.431,A -85,B 0,C 180,E1 -5487.627,E2 -5487.627} C_VEL
LIN {X 0,Y 509.152,Z 785.703,A -85,B 0,C 180,E1 -5488.418,E2 -5488.418} C_VEL
LIN {X 0,Y 509.123,Z 786.493,A -85,B 0,C 180,E1 -5489.209,E2 -5489.209} C_VEL
LIN {X 0,Y 509.142,Z 786.782,A -85,B 0,C 180,E1 -5490,E2 -5490} C_VEL
LIN {X 0,Y 509.124,Z 786.485,A -85,B 0,C 180,E1 -5490.791,E2 -5490.791} C_VEL
LIN {X 0,Y 509.155,Z 785.679,A -85,B 0,C 180,E1 -5491.582,E2 -5491.582} C_VEL
LIN {X 0,Y 509.22,Z 784.389,A -85,B 0,C 180,E1 -5492.373,E2 -5492.373} C_VEL
LIN {X 0,Y 509.288,Z 781.404,A -85,B 0,C 180,E1 -5493.56,E2 -5493.56} C_VEL
LIN {X 0,Y 509.303,Z 778.67,A -85,B 0,C 180,E1 -5494.353,E2 -5494.353} C_VEL
LIN {X 0,Y 509.389,Z 773.357,A -85,B 0,C 180,E1 -5495.542,E2 -5495.542} C_VEL
LIN {X 0,Y 509.505,Z 766.476,A -85,B 0,C 180,E1 -5496.71,E2 -5496.71} C_VEL
LIN {X 0,Y 509.628,Z 758.676,A -85,B 0,C 180,E1 -5497.727,E2 -5497.727} C_VEL
LIN {X 0,Y 509.765,Z 751.145,A -85,B 0,C 180,E1 -5498.523,E2 -5498.523} C_VEL
LIN {X 0,Y 510.037,Z 741.867,A -85,B 0,C 180,E1 -5499.317,E2 -5499.317} C_VEL
LIN {X 0,Y 510.254,Z 731.411,A -85,B 0,C 180,E1 -5500.014,E2 -5500.014} C_VEL
LIN {X 0,Y 510.48,Z 720.308,A -85,B 0,C 180,E1 -5500.56,E2 -5500.56} C_VEL
LIN {X 0,Y 510.646,Z 709.749,A -85,B 0,C 180,E1 -5500.933,E2 -5500.933} C_VEL
LIN {X 0,Y 510.874,Z 698.835,A -85,B 0,C 180,E1 -5501.179,E2 -5501.179} C_VEL
LIN {X 0,Y 510.929,Z 634.519,A -85,B 0,C 180,E1 -5502.101,E2 -5502.101} C_VEL
LIN {X 0,Y 509.845,Z 622.828,A -85,B 0,C 180,E1 -5502.312,E2 -5502.312} C_VEL
LIN {X 0,Y 509.851,Z 620.84,A -85,B 0,C 180,E1 -5502.539,E2 -5502.539} C_VEL
LIN {X 0,Y 510.083,Z 602.756,A -85,B 0,C 180,E1 -5505.176,E2 -5505.176} C_VEL
LIN {X 0,Y 510.369,Z 584.186,A -85,B 0,C 180,E1 -5507.9,E2 -5507.9} C_VEL
LIN {X 0,Y 510.723,Z 563.575,A -85,B 0,C 180,E1 -5510.963,E2 -5510.963} C_VEL
LIN {X 0,Y 511.076,Z 543.992,A -85,B 0,C 180,E1 -5513.932,E2 -5513.932} C_VEL
LIN {X 0,Y 511.444,Z 524.57,A -85,B 0,C 180,E1 -5516.966,E2 -5516.966} C_VEL
LIN {X 0,Y 511.243,Z 519.028,A -85,B 0,C 180,E1 -5517.864,E2 -5517.864} C_VEL
LIN {X 0,Y 509.908,Z 511.903,A -85,B 0,C 180,E1 -5519.124,E2 -5519.124} C_VEL
LIN {X 0,Y 509.862,Z 511.787,A -85,B 0,C 180,E1 -5522.518,E2 -5522.518} C_VEL
LIN {X 0,Y 509.835,Z 511.788,A -85,B 0,C 180,E1 -5525.58,E2 -5525.58} C_VEL
LIN {X 0,Y 509.847,Z 511.786,A -85,B 0,C 180,E1 -5528.337,E2 -5528.337} C_VEL
LIN {X 0,Y 509.853,Z 511.786,A -85,B 0,C 180,E1 -5531.424,E2 -5531.424} C_VEL
LIN {X 0,Y 509.85,Z 511.789,A -85,B 0,C 180,E1 -5534.667,E2 -5534.667} C_VEL
LIN {X 0,Y 509.857,Z 511.781,A -85,B 0,C 180,E1 -5538.102,E2 -5538.102} C_VEL
LIN {X 0,Y 509.87,Z 511.786,A -85,B 0,C 180,E1 -5540.65,E2 -5540.65} C_VEL
LIN {X 0,Y 509.829,Z 511.785,A -85,B 0,C 180,E1 -5543.647,E2 -5543.647} C_VEL
LIN {X 0,Y 509.856,Z 511.787,A -85,B 0,C 180,E1 -5546.539,E2 -5546.539} C_VEL
LIN {X 0,Y 509.842,Z 511.787,A -85,B 0,C 180,E1 -5549.334,E2 -5549.334} C_VEL
LIN {X 0,Y 509.887,Z 511.78,A -85,B 0,C 180,E1 -5552.054,E2 -5552.054} C_VEL
LIN {X 0,Y 509.87,Z 511.785,A -85,B 0,C 180,E1 -5554.704,E2 -5554.704} C_VEL
LIN {X 0,Y 509.846,Z 511.786,A -85,B 0,C 180,E1 -5557.449,E2 -5557.449} C_VEL
LIN {X 0,Y 509.907,Z 511.776,A -85,B 0,C 180,E1 -5559.845,E2 -5559.845} C_VEL
LIN {X 0,Y 509.878,Z 511.786,A -85,B 0,C 180,E1 -5563.175,E2 -5563.175} C_VEL
LIN {X 0,Y 509.854,Z 511.784,A -85,B 0,C 180,E1 -5565.634,E2 -5565.634} C_VEL
LIN {X 0,Y 509.916,Z 511.783,A -85,B 0,C 180,E1 -5568.875,E2 -5568.875} C_VEL
LIN {X 0,Y 509.942,Z 511.774,A -85,B 0,C 180,E1 -5572.079,E2 -5572.079} C_VEL
LIN {X 0,Y 510.001,Z 511.77,A -85,B 0,C 180,E1 -5574.465,E2 -5574.465} C_VEL
LIN {X 0,Y 510.047,Z 511.761,A -85,B 0,C 180,E1 -5577.631,E2 -5577.631} C_VEL
LIN {X 0,Y 510.057,Z 511.767,A -85,B 0,C 180,E1 -5580.79,E2 -5580.79} C_VEL
LIN {X 0,Y 509.952,Z 511.777,A -85,B 0,C 180,E1 -5583.16,E2 -5583.16} C_VEL
LIN {X 0,Y 509.968,Z 511.777,A -85,B 0,C 180,E1 -5586.33,E2 -5586.33} C_VEL
LIN {X 0,Y 509.978,Z 512.099,A -85,B 0,C 180,E1 -5586.694,E2 -5586.694} C_VEL
LIN {X 0,Y 510.296,Z 513.352,A -85,B 0,C 180,E1 -5586.799,E2 -5586.799} C_VEL
LIN {X 0,Y 511.659,Z 517.922,A -85,B 0,C 180,E1 -5586.905,E2 -5586.905} C_VEL
LIN {X 0,Y 511.58,Z 541.849,A -85,B 0,C 180,E1 -5587.261,E2 -5587.261} C_VEL
LIN {X 0,Y 511.52,Z 555.304,A -85,B 0,C 180,E1 -5587.628,E2 -5587.628} C_VEL
LIN {X 0,Y 511.392,Z 567.054,A -85,B 0,C 180,E1 -5588.102,E2 -5588.102} C_VEL
LIN {X 0,Y 511.213,Z 578.089,A -85,B 0,C 180,E1 -5588.698,E2 -5588.698} C_VEL
LIN {X 0,Y 510.951,Z 589.584,A -85,B 0,C 180,E1 -5589.501,E2 -5589.501} C_VEL
LIN {X 0,Y 510.624,Z 599.934,A -85,B 0,C 180,E1 -5590.408,E2 -5590.408} C_VEL
LIN {X 0,Y 510.384,Z 608.333,A -85,B 0,C 180,E1 -5591.316,E2 -5591.316} C_VEL
LIN {X 0,Y 510.146,Z 617.372,A -85,B 0,C 180,E1 -5592.532,E2 -5592.532} C_VEL
LIN {X 0,Y 509.928,Z 624.646,A -85,B 0,C 180,E1 -5593.754,E2 -5593.754} C_VEL
LIN {X 0,Y 509.767,Z 629.541,A -85,B 0,C 180,E1 -5594.777,E2 -5594.777} C_VEL
LIN {X 0,Y 509.626,Z 634.261,A -85,B 0,C 180,E1 -5596.011,E2 -5596.011} C_VEL
LIN {X 0,Y 509.539,Z 637.824,A -85,B 0,C 180,E1 -5597.251,E2 -5597.251} C_VEL
LIN {X 0,Y 509.451,Z 640.326,A -85,B 0,C 180,E1 -5598.499,E2 -5598.499} C_VEL
LIN {X 0,Y 509.415,Z 641.411,A -85,B 0,C 180,E1 -5599.336,E2 -5599.336} C_VEL
LIN {X 0,Y 509.38,Z 642.108,A -85,B 0,C 180,E1 -5600.251,E2 -5600.251} C_VEL
LIN {X 0,Y 509.374,Z 642.304,A -85,B 0,C 180,E1 -5601.023,E2 -5601.023} C_VEL
LIN {X 0,Y 509.386,Z 641.666,A -85,B 0,C 180,E1 -5602.426,E2 -5602.426} C_VEL
LIN {X 0,Y 509.441,Z 640.223,A -85,B 0,C 180,E1 -5603.583,E2 -5603.583} C_VEL
LIN {X 0,Y 509.542,Z 637.551,A -85,B 0,C 180,E1 -5604.878,E2 -5604.878} C_VEL
LIN {X 0,Y 509.651,Z 633.185,A -85,B 0,C 180,E1 -5606.322,E2 -5606.322} C_VEL
LIN {X 0,Y 509.773,Z 627.409,A -85,B 0,C 180,E1 -5607.73,E2 -5607.73} C_VEL
LIN {X 0,Y 509.98,Z 620.198,A -85,B 0,C 180,E1 -5609.064,E2 -5609.064} C_VEL
LIN {X 0,Y 510.22,Z 612.635,A -85,B 0,C 180,E1 -5610.183,E2 -5610.183} C_VEL
LIN {X 0,Y 510.517,Z 603.188,A -85,B 0,C 180,E1 -5611.311,E2 -5611.311} C_VEL
LIN {X 0,Y 510.78,Z 592.395,A -85,B 0,C 180,E1 -5612.337,E2 -5612.337} C_VEL
LIN {X 0,Y 511.068,Z 582.093,A -85,B 0,C 180,E1 -5613.12,E2 -5613.12} C_VEL
LIN {X 0,Y 511.33,Z 570.263,A -85,B 0,C 180,E1 -5613.825,E2 -5613.825} C_VEL
LIN {X 0,Y 511.52,Z 557.817,A -85,B 0,C 180,E1 -5614.382,E2 -5614.382} C_VEL
LIN {X 0,Y 511.635,Z 544.878,A -85,B 0,C 180,E1 -5614.787,E2 -5614.787} C_VEL
LIN {X 0,Y 511.689,Z 529.452,A -85,B 0,C 180,E1 -5615.063,E2 -5615.063} C_VEL
LIN {X 0,Y 511.669,Z 517.77,A -85,B 0,C 180,E1 -5615.23,E2 -5615.23} C_VEL
LIN {X 0,Y 510.401,Z 513.803,A -85,B 0,C 180,E1 -5615.324,E2 -5615.324} C_VEL
LIN {X 0,Y 509.62,Z 512.589,A -85,B 0,C 180,E1 -5615.443,E2 -5615.443} C_VEL
LIN {X 0,Y 508.356,Z 512.057,A -85,B 0,C 180,E1 -5615.712,E2 -5615.712} C_VEL
LIN {X 0,Y 505.264,Z 512.362,A -85,B 0,C 180,E1 -5616.711,E2 -5616.711} C_VEL
LIN {X 0,Y 503.83,Z 512.853,A -85,B 0,C 180,E1 -5617.474,E2 -5617.474} C_VEL
LIN {X 0,Y 502.964,Z 512.745,A -85,B 0,C 180,E1 -5618.255,E2 -5618.255} C_VEL
LIN {X 0,Y 502.791,Z 512.668,A -85,B 0,C 180,E1 -5618.779,E2 -5618.779} C_VEL
LIN {X 0,Y 502.826,Z 512.66,A -85,B 0,C 180,E1 -5622.137,E2 -5622.137} C_VEL
LIN {X 0,Y 502.798,Z 512.669,A -85,B 0,C 180,E1 -5625.469,E2 -5625.469} C_VEL
LIN {X 0,Y 502.828,Z 512.66,A -85,B 0,C 180,E1 -5627.865,E2 -5627.865} C_VEL
LIN {X 0,Y 502.809,Z 512.664,A -85,B 0,C 180,E1 -5631.026,E2 -5631.026} C_VEL
LIN {X 0,Y 502.774,Z 512.665,A -85,B 0,C 180,E1 -5634.17,E2 -5634.17} C_VEL
LIN {X 0,Y 502.833,Z 512.66,A -85,B 0,C 180,E1 -5636.994,E2 -5636.994} C_VEL
LIN {X 0,Y 502.816,Z 512.661,A -85,B 0,C 180,E1 -5640.066,E2 -5640.066} C_VEL
LIN {X 0,Y 502.836,Z 512.656,A -85,B 0,C 180,E1 -5642.534,E2 -5642.534} C_VEL
LIN {X 0,Y 502.829,Z 512.663,A -85,B 0,C 180,E1 -5645.3,E2 -5645.3} C_VEL
LIN {X 0,Y 502.783,Z 512.668,A -85,B 0,C 180,E1 -5647.827,E2 -5647.827} C_VEL
LIN {X 0,Y 502.827,Z 512.658,A -85,B 0,C 180,E1 -5650.401,E2 -5650.401} C_VEL
LIN {X 0,Y 502.822,Z 512.659,A -85,B 0,C 180,E1 -5652.932,E2 -5652.932} C_VEL
LIN {X 0,Y 502.849,Z 512.661,A -85,B 0,C 180,E1 -5655.43,E2 -5655.43} C_VEL
LIN {X 0,Y 502.882,Z 512.651,A -85,B 0,C 180,E1 -5658.717,E2 -5658.717} C_VEL
LIN {X 0,Y 502.906,Z 512.653,A -85,B 0,C 180,E1 -5661.967,E2 -5661.967} C_VEL
LIN {X 0,Y 502.93,Z 512.646,A -85,B 0,C 180,E1 -5664.387,E2 -5664.387} C_VEL
LIN {X 0,Y 503.029,Z 512.64,A -85,B 0,C 180,E1 -5667.598,E2 -5667.598} C_VEL
LIN {X 0,Y 503.033,Z 512.637,A -85,B 0,C 180,E1 -5670,E2 -5670} C_VEL
LIN {X 0,Y 503.029,Z 512.634,A -85,B 0,C 180,E1 -5672.402,E2 -5672.402} C_VEL
LIN {X 0,Y 502.931,Z 512.651,A -85,B 0,C 180,E1 -5675.613,E2 -5675.613} C_VEL
LIN {X 0,Y 502.872,Z 512.652,A -85,B 0,C 180,E1 -5678.843,E2 -5678.843} C_VEL
LIN {X 0,Y 502.851,Z 512.66,A -85,B 0,C 180,E1 -5682.101,E2 -5682.101} C_VEL
LIN {X 0,Y 502.853,Z 512.657,A -85,B 0,C 180,E1 -5685.399,E2 -5685.399} C_VEL
LIN {X 0,Y 502.85,Z 512.66,A -85,B 0,C 180,E1 -5688.122,E2 -5688.122} C_VEL
LIN {X 0,Y 502.832,Z 512.658,A -85,B 0,C 180,E1 -5690.536,E2 -5690.536} C_VEL
LIN {X 0,Y 502.791,Z 512.662,A -85,B 0,C 180,E1 -5693.04,E2 -5693.04} C_VEL
LIN {X 0,Y 502.824,Z 512.663,A -85,B 0,C 180,E1 -5695.676,E2 -5695.676} C_VEL
LIN {X 0,Y 502.842,Z 512.659,A -85,B 0,C 180,E1 -5698.372,E2 -5698.372} C_VEL
LIN {X 0,Y 502.794,Z 512.664,A -85,B 0,C 180,E1 -5701.498,E2 -5701.498} C_VEL
LIN {X 0,Y 502.804,Z 512.67,A -85,B 0,C 180,E1 -5703.993,E2 -5703.993} C_VEL
LIN {X 0,Y 502.777,Z 512.664,A -85,B 0,C 180,E1 -5707.177,E2 -5707.177} C_VEL
LIN {X 0,Y 502.821,Z 512.667,A -85,B 0,C 180,E1 -5710.011,E2 -5710.011} C_VEL
LIN {X 0,Y 502.822,Z 512.666,A -85,B 0,C 180,E1 -5712.201,E2 -5712.201} C_VEL
LIN {X 0,Y 502.798,Z 512.662,A -85,B 0,C 180,E1 -5715.467,E2 -5715.467} C_VEL
LIN {X 0,Y 502.817,Z 512.659,A -85,B 0,C 180,E1 -5718.933,E2 -5718.933} C_VEL
LIN {X 0,Y 502.79,Z 512.67,A -85,B 0,C 180,E1 -5722.045,E2 -5722.045} C_VEL
LIN {X 0,Y 502.805,Z 512.661,A -85,B 0,C 180,E1 -5725.034,E2 -5725.034} C_VEL
LIN {X 0,Y 502.783,Z 512.668,A -85,B 0,C 180,E1 -5727.915,E2 -5727.915} C_VEL
LIN {X 0,Y 502.834,Z 512.66,A -85,B 0,C 180,E1 -5730.712,E2 -5730.712} C_VEL
LIN {X 0,Y 502.875,Z 512.652,A -85,B 0,C 180,E1 -5733.434,E2 -5733.434} C_VEL
LIN {X 0,Y 502.785,Z 512.669,A -85,B 0,C 180,E1 -5736.086,E2 -5736.086} C_VEL
LIN {X 0,Y 502.777,Z 512.668,A -85,B 0,C 180,E1 -5738.688,E2 -5738.688} C_VEL
LIN {X 0,Y 502.823,Z 512.658,A -85,B 0,C 180,E1 -5741.248,E2 -5741.248} C_VEL
LIN {X 0,Y 502.816,Z 512.661,A -85,B 0,C 180,E1 -5743.767,E2 -5743.767} C_VEL
LIN {X 0,Y 502.823,Z 512.666,A -85,B 0,C 180,E1 -5746.254,E2 -5746.254} C_VEL
LIN {X 0,Y 502.884,Z 512.655,A -85,B 0,C 180,E1 -5748.717,E2 -5748.717} C_VEL
LIN {X 0,Y 502.894,Z 512.652,A -85,B 0,C 180,E1 -5751.966,E2 -5751.966} C_VEL
LIN {X 0,Y 502.95,Z 512.651,A -85,B 0,C 180,E1 -5754.386,E2 -5754.386} C_VEL
LIN {X 0,Y 503.016,Z 512.634,A -85,B 0,C 180,E1 -5757.597,E2 -5757.597} C_VEL
LIN {X 0,Y 503.017,Z 512.636,A -85,B 0,C 180,E1 -5760,E2 -5760} C_VEL
LIN {X 0,Y 503.016,Z 512.642,A -85,B 0,C 180,E1 -5762.402,E2 -5762.402} C_VEL
LIN {X 0,Y 502.93,Z 512.645,A -85,B 0,C 180,E1 -5765.613,E2 -5765.613} C_VEL
LIN {X 0,Y 502.893,Z 512.652,A -85,B 0,C 180,E1 -5768.033,E2 -5768.033} C_VEL
LIN {X 0,Y 502.868,Z 512.653,A -85,B 0,C 180,E1 -5771.283,E2 -5771.283} C_VEL
LIN {X 0,Y 502.842,Z 512.665,A -85,B 0,C 180,E1 -5774.571,E2 -5774.571} C_VEL
LIN {X 0,Y 502.853,Z 512.655,A -85,B 0,C 180,E1 -5777.907,E2 -5777.907} C_VEL
LIN {X 0,Y 502.82,Z 512.666,A -85,B 0,C 180,E1 -5780.536,E2 -5780.536} C_VEL
LIN {X 0,Y 502.788,Z 512.666,A -85,B 0,C 180,E1 -5783.041,E2 -5783.041} C_VEL
LIN {X 0,Y 502.833,Z 512.657,A -85,B 0,C 180,E1 -5785.676,E2 -5785.676} C_VEL
LIN {X 0,Y 502.834,Z 512.661,A -85,B 0,C 180,E1 -5788.373,E2 -5788.373} C_VEL
LIN {X 0,Y 502.789,Z 512.663,A -85,B 0,C 180,E1 -5791.5,E2 -5791.5} C_VEL
LIN {X 0,Y 502.8,Z 512.665,A -85,B 0,C 180,E1 -5794.445,E2 -5794.445} C_VEL
LIN {X 0,Y 502.774,Z 512.668,A -85,B 0,C 180,E1 -5797.179,E2 -5797.179} C_VEL
LIN {X 0,Y 502.782,Z 512.664,A -85,B 0,C 180,E1 -5800.016,E2 -5800.016} C_VEL
LIN {X 0,Y 502.796,Z 512.663,A -85,B 0,C 180,E1 -5802.2,E2 -5802.2} C_VEL
LIN {X 0,Y 502.795,Z 512.663,A -85,B 0,C 180,E1 -5805.469,E2 -5805.469} C_VEL
LIN {X 0,Y 502.825,Z 512.658,A -85,B 0,C 180,E1 -5807.865,E2 -5807.865} C_VEL
LIN {X 0,Y 502.799,Z 512.669,A -85,B 0,C 180,E1 -5811.025,E2 -5811.025} C_VEL
LIN {X 0,Y 502.779,Z 512.666,A -85,B 0,C 180,E1 -5814.168,E2 -5814.168} C_VEL
LIN {X 0,Y 502.83,Z 512.666,A -85,B 0,C 180,E1 -5816.994,E2 -5816.994} C_VEL
LIN {X 0,Y 502.847,Z 512.704,A -85,B 0,C 180,E1 -5819.923,E2 -5819.923} C_VEL
LIN {X 0,Y 503.205,Z 514.583,A -85,B 0,C 180,E1 -5820.327,E2 -5820.327} C_VEL
LIN {X 0,Y 505.214,Z 525.233,A -85,B 0,C 180,E1 -5822.225,E2 -5822.225} C_VEL
LIN {X 0,Y 504.691,Z 541.189,A -85,B 0,C 180,E1 -5824.843,E2 -5824.843} C_VEL
LIN {X 0,Y 504.124,Z 560.151,A -85,B 0,C 180,E1 -5827.889,E2 -5827.889} C_VEL
LIN {X 0,Y 503.614,Z 581.551,A -85,B 0,C 180,E1 -5831.279,E2 -5831.279} C_VEL
LIN {X 0,Y 503.097,Z 606.397,A -85,B 0,C 180,E1 -5835.023,E2 -5835.023} C_VEL
LIN {X 0,Y 502.808,Z 622.406,A -85,B 0,C 180,E1 -5837.462,E2 -5837.462} C_VEL
LIN {X 0,Y 504.233,Z 637.158,A -85,B 0,C 180,E1 -5837.736,E2 -5837.736} C_VEL
LIN {X 0,Y 503.893,Z 701.805,A -85,B 0,C 180,E1 -5838.716,E2 -5838.716} C_VEL
LIN {X 0,Y 503.595,Z 713.677,A -85,B 0,C 180,E1 -5839.039,E2 -5839.039} C_VEL
LIN {X 0,Y 503.384,Z 725.398,A -85,B 0,C 180,E1 -5839.543,E2 -5839.543} C_VEL
LIN {X 0,Y 503.104,Z 735.641,A -85,B 0,C 180,E1 -5840.147,E2 -5840.147} C_VEL
LIN {X 0,Y 502.916,Z 745.009,A -85,B 0,C 180,E1 -5840.854,E2 -5840.854} C_VEL
LIN {X 0,Y 502.643,Z 754.452,A -85,B 0,C 180,E1 -5841.76,E2 -5841.76} C_VEL
LIN {X 0,Y 502.457,Z 762.66,A -85,B 0,C 180,E1 -5842.768,E2 -5842.768} C_VEL
LIN {X 0,Y 502.388,Z 769.228,A -85,B 0,C 180,E1 -5843.776,E2 -5843.776} C_VEL
LIN {X 0,Y 502.229,Z 774.455,A -85,B 0,C 180,E1 -5844.781,E2 -5844.781} C_VEL
LIN {X 0,Y 502.26,Z 779.284,A -85,B 0,C 180,E1 -5845.988,E2 -5845.988} C_VEL
LIN {X 0,Y 502.195,Z 781.668,A -85,B 0,C 180,E1 -5846.791,E2 -5846.791} C_VEL
LIN {X 0,Y 502.167,Z 783.464,A -85,B 0,C 180,E1 -5847.594,E2 -5847.594} C_VEL
LIN {X 0,Y 502.113,Z 784.734,A -85,B 0,C 180,E1 -5848.396,E2 -5848.396} C_VEL
LIN {X 0,Y 502.088,Z 785.518,A -85,B 0,C 180,E1 -5849.198,E2 -5849.198} C_VEL
LIN {X 0,Y 502.13,Z 785.795,A -85,B 0,C 180,E1 -5850,E2 -5850} C_VEL
LIN {X 0,Y 502.091,Z 785.501,A -85,B 0,C 180,E1 -5850.802,E2 -5850.802} C_VEL
LIN {X 0,Y 502.12,Z 784.684,A -85,B 0,C 180,E1 -5851.604,E2 -5851.604} C_VEL
LIN {X 0,Y 502.178,Z 783.38,A -85,B 0,C 180,E1 -5852.406,E2 -5852.406} C_VEL
LIN {X 0,Y 502.247,Z 780.38,A -85,B 0,C 180,E1 -5853.61,E2 -5853.61} C_VEL
LIN {X 0,Y 502.236,Z 777.625,A -85,B 0,C 180,E1 -5854.414,E2 -5854.414} C_VEL
LIN {X 0,Y 502.34,Z 772.296,A -85,B 0,C 180,E1 -5855.62,E2 -5855.62} C_VEL
LIN {X 0,Y 502.449,Z 765.11,A -85,B 0,C 180,E1 -5856.842,E2 -5856.842} C_VEL
LIN {X 0,Y 502.576,Z 757.557,A -85,B 0,C 180,E1 -5857.836,E2 -5857.836} C_VEL
LIN {X 0,Y 502.801,Z 748.979,A -85,B 0,C 180,E1 -5858.743,E2 -5858.743} C_VEL
LIN {X 0,Y 503.008,Z 739.373,A -85,B 0,C 180,E1 -5859.55,E2 -5859.55} C_VEL
LIN {X 0,Y 503.238,Z 728.4,A -85,B 0,C 180,E1 -5860.257,E2 -5860.257} C_VEL
LIN {X 0,Y 503.493,Z 717.918,A -85,B 0,C 180,E1 -5860.76,E2 -5860.76} C_VEL
LIN {X 0,Y 503.696,Z 706.883,A -85,B 0,C 180,E1 -5861.137,E2 -5861.137} C_VEL
LIN {X 0,Y 503.94,Z 693.558,A -85,B 0,C 180,E1 -5861.401,E2 -5861.401} C_VEL
LIN {X 0,Y 503.975,Z 635.033,A -85,B 0,C 180,E1 -5862.256,E2 -5862.256} C_VEL
LIN {X 0,Y 502.763,Z 620.912,A -85,B 0,C 180,E1 -5862.526,E2 -5862.526} C_VEL
LIN {X 0,Y 503.013,Z 604.147,A -85,B 0,C 180,E1 -5864.979,E2 -5864.979} C_VEL
LIN {X 0,Y 503.296,Z 582.7,A -85,B 0,C 180,E1 -5868.182,E2 -5868.182} C_VEL
LIN {X 0,Y 503.717,Z 562.318,A -85,B 0,C 180,E1 -5871.269,E2 -5871.269} C_VEL
LIN {X 0,Y 504.104,Z 542.843,A -85,B 0,C 180,E1 -5874.284,E2 -5874.284} C_VEL
LIN {X 0,Y 504.46,Z 525.219,A -85,B 0,C 180,E1 -5877.097,E2 -5877.097} C_VEL
LIN {X 0,Y 504.347,Z 520.789,A -85,B 0,C 180,E1 -5877.827,E2 -5877.827} C_VEL
LIN {X 0,Y 502.874,Z 512.874,A -85,B 0,C 180,E1 -5879.229,E2 -5879.229} C_VEL
LIN {X 0,Y 502.793,Z 512.667,A -85,B 0,C 180,E1 -5881.499,E2 -5881.499} C_VEL
LIN {X 0,Y 502.8,Z 512.667,A -85,B 0,C 180,E1 -5884.444,E2 -5884.444} C_VEL
LIN {X 0,Y 502.776,Z 512.672,A -85,B 0,C 180,E1 -5887.178,E2 -5887.178} C_VEL
LIN {X 0,Y 502.783,Z 512.664,A -85,B 0,C 180,E1 -5890.014,E2 -5890.014} C_VEL
LIN {X 0,Y 502.797,Z 512.663,A -85,B 0,C 180,E1 -5892.199,E2 -5892.199} C_VEL
LIN {X 0,Y 502.794,Z 512.665,A -85,B 0,C 180,E1 -5895.468,E2 -5895.468} C_VEL
LIN {X 0,Y 502.823,Z 512.657,A -85,B 0,C 180,E1 -5897.864,E2 -5897.864} C_VEL
LIN {X 0,Y 502.815,Z 512.665,A -85,B 0,C 180,E1 -5901.025,E2 -5901.025} C_VEL
LIN {X 0,Y 502.779,Z 512.663,A -85,B 0,C 180,E1 -5904.166,E2 -5904.166} C_VEL
LIN {X 0,Y 502.825,Z 512.664,A -85,B 0,C 180,E1 -5906.993,E2 -5906.993} C_VEL
LIN {X 0,Y 502.822,Z 512.659,A -85,B 0,C 180,E1 -5910.061,E2 -5910.061} C_VEL
LIN {X 0,Y 502.827,Z 512.663,A -85,B 0,C 180,E1 -5912.533,E2 -5912.533} C_VEL
LIN {X 0,Y 502.82,Z 512.663,A -85,B 0,C 180,E1 -5915.298,E2 -5915.298} C_VEL
LIN {X 0,Y 502.784,Z 512.664,A -85,B 0,C 180,E1 -5917.827,E2 -5917.827} C_VEL
LIN {X 0,Y 502.817,Z 512.661,A -85,B 0,C 180,E1 -5920.4,E2 -5920.4} C_VEL
LIN {X 0,Y 502.827,Z 512.666,A -85,B 0,C 180,E1 -5922.932,E2 -5922.932} C_VEL
LIN {X 0,Y 502.835,Z 512.66,A -85,B 0,C 180,E1 -5925.429,E2 -5925.429} C_VEL
LIN {X 0,Y 502.885,Z 512.659,A -85,B 0,C 180,E1 -5928.717,E2 -5928.717} C_VEL
LIN {X 0,Y 502.893,Z 512.652,A -85,B 0,C 180,E1 -5931.967,E2 -5931.967} C_VEL
LIN {X 0,Y 502.953,Z 512.647,A -85,B 0,C 180,E1 -5934.387,E2 -5934.387} C_VEL
LIN {X 0,Y 503.017,Z 512.637,A -85,B 0,C 180,E1 -5937.598,E2 -5937.598} C_VEL
LIN {X 0,Y 503.017,Z 512.637,A -85,B 0,C 180,E1 -5940,E2 -5940} C_VEL
LIN {X 0,Y 503.016,Z 512.64,A -85,B 0,C 180,E1 -5942.403,E2 -5942.403} C_VEL
LIN {X 0,Y 502.953,Z 512.65,A -85,B 0,C 180,E1 -5945.614,E2 -5945.614} C_VEL
LIN {X 0,Y 502.943,Z 512.886,A -85,B 0,C 180,E1 -5946.493,E2 -5946.493} C_VEL
LIN {X 0,Y 503.207,Z 514.11,A -85,B 0,C 180,E1 -5946.619,E2 -5946.619} C_VEL
LIN {X 0,Y 504.763,Z 519.59,A -85,B 0,C 180,E1 -5946.745,E2 -5946.745} C_VEL
LIN {X 0,Y 504.699,Z 543.203,A -85,B 0,C 180,E1 -5947.104,E2 -5947.104} C_VEL
LIN {X 0,Y 504.637,Z 556.654,A -85,B 0,C 180,E1 -5947.477,E2 -5947.477} C_VEL
LIN {X 0,Y 504.46,Z 569.403,A -85,B 0,C 180,E1 -5948.009,E2 -5948.009} C_VEL
LIN {X 0,Y 504.229,Z 581.878,A -85,B 0,C 180,E1 -5948.725,E2 -5948.725} C_VEL
LIN {X 0,Y 503.996,Z 592.778,A -85,B 0,C 180,E1 -5949.532,E2 -5949.532} C_VEL
LIN {X 0,Y 503.679,Z 602.657,A -85,B 0,C 180,E1 -5950.451,E2 -5950.451} C_VEL
LIN {X 0,Y 503.403,Z 611.488,A -85,B 0,C 180,E1 -5951.464,E2 -5951.464} C_VEL
LIN {X 0,Y 503.112,Z 620.129,A -85,B 0,C 180,E1 -5952.69,E2 -5952.69} C_VEL
LIN {X 0,Y 502.906,Z 627.116,A -85,B 0,C 180,E1 -5953.95,E2 -5953.95} C_VEL
LIN {X 0,Y 502.709,Z 633.392,A -85,B 0,C 180,E1 -5955.404,E2 -5955.404} C_VEL
LIN {X 0,Y 502.566,Z 637.448,A -85,B 0,C 180,E1 -5956.659,E2 -5956.659} C_VEL
LIN {X 0,Y 502.477,Z 640.525,A -85,B 0,C 180,E1 -5957.997,E2 -5957.997} C_VEL
LIN {X 0,Y 502.377,Z 642.711,A -85,B 0,C 180,E1 -5959.618,E2 -5959.618} C_VEL
LIN {X 0,Y 502.371,Z 643.22,A -85,B 0,C 180,E1 -5960.472,E2 -5960.472} C_VEL
LIN {X 0,Y 502.345,Z 643.254,A -85,B 0,C 180,E1 -5961.331,E2 -5961.331} C_VEL
LIN {X 0,Y 502.384,Z 642.512,A -85,B 0,C 180,E1 -5962.591,E2 -5962.591} C_VEL
LIN {X 0,Y 502.428,Z 640.648,A -85,B 0,C 180,E1 -5963.933,E2 -5963.933} C_VEL
LIN {X 0,Y 502.547,Z 637.695,A -85,B 0,C 180,E1 -5965.248,E2 -5965.248} C_VEL
LIN {X 0,Y 502.671,Z 633.502,A -85,B 0,C 180,E1 -5966.578,E2 -5966.578} C_VEL
LIN {X 0,Y 502.793,Z 628.012,A -85,B 0,C 180,E1 -5967.889,E2 -5967.889} C_VEL
LIN {X 0,Y 503.029,Z 620.495,A -85,B 0,C 180,E1 -5969.275,E2 -5969.275} C_VEL
LIN {X 0,Y 503.309,Z 612.77,A -85,B 0,C 180,E1 -5970.41,E2 -5970.41} C_VEL
LIN {X 0,Y 503.595,Z 604.138,A -85,B 0,C 180,E1 -5971.44,E2 -5971.44} C_VEL
LIN {X 0,Y 503.843,Z 594.654,A -85,B 0,C 180,E1 -5972.364,E2 -5972.364} C_VEL
LIN {X 0,Y 504.157,Z 583.475,A -85,B 0,C 180,E1 -5973.24,E2 -5973.24} C_VEL
LIN {X 0,Y 504.428,Z 572.247,A -85,B 0,C 180,E1 -5973.93,E2 -5973.93} C_VEL
LIN {X 0,Y 504.631,Z 559.514,A -85,B 0,C 180,E1 -5974.518,E2 -5974.518} C_VEL
LIN {X 0,Y 504.769,Z 546.774,A -85,B 0,C 180,E1 -5974.932,E2 -5974.932} C_VEL
LIN {X 0,Y 504.806,Z 533.413,A -85,B 0,C 180,E1 -5975.191,E2 -5975.191} C_VEL
LIN {X 0,Y 504.727,Z 518.902,A -85,B 0,C 180,E1 -5975.405,E2 -5975.405} C_VEL
LIN {X 0,Y 502.996,Z 513.539,A -85,B 0,C 180,E1 -5975.558,E2 -5975.558} C_VEL
LIN {X 0,Y 502.827,Z 512.721,A -85,B 0,C 180,E1 -5975.731,E2 -5975.731} C_VEL
LIN {X 0,Y 502.791,Z 512.668,A -85,B 0,C 180,E1 -5978.779,E2 -5978.779} C_VEL
LIN {X 0,Y 502.141,Z 512.753,A -85,B 0,C 180,E1 -5979.448,E2 -5979.448} C_VEL
LIN {X 0,Y 499.292,Z 513.106,A -85,B 0,C 180,E1 -5980.534,E2 -5980.534} C_VEL
LIN {X 0,Y 496.87,Z 513.409,A -85,B 0,C 180,E1 -5981.409,E2 -5981.409} C_VEL
LIN {X 0,Y 495.826,Z 513.532,A -85,B 0,C 180,E1 -5982.085,E2 -5982.085} C_VEL
LIN {X 0,Y 495.739,Z 513.542,A -85,B 0,C 180,E1 -5982.314,E2 -5982.314} C_VEL
LIN {X 0,Y 495.747,Z 513.545,A -85,B 0,C 180,E1 -5985.14,E2 -5985.14} C_VEL
LIN {X 0,Y 495.777,Z 513.536,A -85,B 0,C 180,E1 -5988.222,E2 -5988.222} C_VEL
LIN {X 0,Y 495.768,Z 513.543,A -85,B 0,C 180,E1 -5991.232,E2 -5991.232} C_VEL
LIN {X 0,Y 495.747,Z 513.54,A -85,B 0,C 180,E1 -5994.463,E2 -5994.463} C_VEL
LIN {X 0,Y 495.768,Z 513.545,A -85,B 0,C 180,E1 -5997.407,E2 -5997.407} C_VEL
LIN {X 0,Y 495.767,Z 513.538,A -85,B 0,C 180,E1 -6000.255,E2 -6000.255} C_VEL
LIN {X 0,Y 495.826,Z 513.535,A -85,B 0,C 180,E1 -6003.252,E2 -6003.252} C_VEL
LIN {X 0,Y 495.75,Z 513.546,A -85,B 0,C 180,E1 -6005.726,E2 -6005.726} C_VEL
LIN {X 0,Y 495.745,Z 513.54,A -85,B 0,C 180,E1 -6008.372,E2 -6008.372} C_VEL
LIN {X 0,Y 495.785,Z 513.536,A -85,B 0,C 180,E1 -6010.972,E2 -6010.972} C_VEL
LIN {X 0,Y 495.811,Z 513.532,A -85,B 0,C 180,E1 -6014.377,E2 -6014.377} C_VEL
LIN {X 0,Y 495.815,Z 513.539,A -85,B 0,C 180,E1 -6017.724,E2 -6017.724} C_VEL
LIN {X 0,Y 495.843,Z 513.529,A -85,B 0,C 180,E1 -6021.031,E2 -6021.031} C_VEL
LIN {X 0,Y 495.885,Z 513.524,A -85,B 0,C 180,E1 -6024.307,E2 -6024.307} C_VEL
LIN {X 0,Y 495.997,Z 513.515,A -85,B 0,C 180,E1 -6027.564,E2 -6027.564} C_VEL
LIN {X 0,Y 495.988,Z 513.51,A -85,B 0,C 180,E1 -6030.812,E2 -6030.812} C_VEL
LIN {X 0,Y 495.998,Z 513.509,A -85,B 0,C 180,E1 -6032.436,E2 -6032.436} C_VEL
LIN {X 0,Y 495.886,Z 513.53,A -85,B 0,C 180,E1 -6035.694,E2 -6035.694} C_VEL
LIN {X 0,Y 495.842,Z 513.528,A -85,B 0,C 180,E1 -6038.97,E2 -6038.97} C_VEL
LIN {X 0,Y 495.833,Z 513.535,A -85,B 0,C 180,E1 -6042.035,E2 -6042.035} C_VEL
LIN {X 0,Y 495.828,Z 513.533,A -85,B 0,C 180,E1 -6045.451,E2 -6045.451} C_VEL
LIN {X 0,Y 495.811,Z 513.536,A -85,B 0,C 180,E1 -6048.247,E2 -6048.247} C_VEL
LIN {X 0,Y 495.778,Z 513.536,A -85,B 0,C 180,E1 -6050.756,E2 -6050.756} C_VEL
LIN {X 0,Y 495.746,Z 513.542,A -85,B 0,C 180,E1 -6053.387,E2 -6053.387} C_VEL
LIN {X 0,Y 495.826,Z 513.53,A -85,B 0,C 180,E1 -6056.749,E2 -6056.749} C_VEL
LIN {X 0,Y 495.768,Z 513.543,A -85,B 0,C 180,E1 -6059.746,E2 -6059.746} C_VEL
LIN {X 0,Y 495.768,Z 513.539,A -85,B 0,C 180,E1 -6062.594,E2 -6062.594} C_VEL
LIN {X 0,Y 495.748,Z 513.542,A -85,B 0,C 180,E1 -6065.537,E2 -6065.537} C_VEL
LIN {X 0,Y 495.768,Z 513.538,A -85,B 0,C 180,E1 -6068.768,E2 -6068.768} C_VEL
LIN {X 0,Y 495.781,Z 513.54,A -85,B 0,C 180,E1 -6071.777,E2 -6071.777} C_VEL
LIN {X 0,Y 495.747,Z 513.54,A -85,B 0,C 180,E1 -6075.138,E2 -6075.138} C_VEL
LIN {X 0,Y 495.755,Z 513.547,A -85,B 0,C 180,E1 -6078.218,E2 -6078.218} C_VEL
LIN {X 0,Y 495.747,Z 513.54,A -85,B 0,C 180,E1 -6081.408,E2 -6081.408} C_VEL
LIN {X 0,Y 495.754,Z 513.544,A -85,B 0,C 180,E1 -6084.462,E2 -6084.462} C_VEL
LIN {X 0,Y 495.765,Z 513.538,A -85,B 0,C 180,E1 -6087.405,E2 -6087.405} C_VEL
LIN {X 0,Y 495.777,Z 513.545,A -85,B 0,C 180,E1 -6090.254,E2 -6090.254} C_VEL
LIN {X 0,Y 495.828,Z 513.53,A -85,B 0,C 180,E1 -6093.247,E2 -6093.247} C_VEL
LIN {X 0,Y 495.746,Z 513.542,A -85,B 0,C 180,E1 -6095.724,E2 -6095.724} C_VEL
LIN {X 0,Y 495.736,Z 513.549,A -85,B 0,C 180,E1 -6098.37,E2 -6098.37} C_VEL
LIN {X 0,Y 495.778,Z 513.537,A -85,B 0,C 180,E1 -6100.971,E2 -6100.971} C_VEL
LIN {X 0,Y 495.773,Z 513.537,A -85,B 0,C 180,E1 -6103.529,E2 -6103.529} C_VEL
LIN {X 0,Y 495.786,Z 513.539,A -85,B 0,C 180,E1 -6106.055,E2 -6106.055} C_VEL
LIN {X 0,Y 495.859,Z 513.532,A -85,B 0,C 180,E1 -6108.555,E2 -6108.555} C_VEL
LIN {X 0,Y 495.865,Z 513.527,A -85,B 0,C 180,E1 -6111.852,E2 -6111.852} C_VEL
LIN {X 0,Y 495.905,Z 513.527,A -85,B 0,C 180,E1 -6114.306,E2 -6114.306} C_VEL
LIN {X 0,Y 495.985,Z 513.51,A -85,B 0,C 180,E1 -6117.563,E2 -6117.563} C_VEL
LIN {X 0,Y 495.989,Z 513.512,A -85,B 0,C 180,E1 -6120,E2 -6120} C_VEL
LIN {X 0,Y 495.985,Z 513.518,A -85,B 0,C 180,E1 -6122.436,E2 -6122.436} C_VEL
LIN {X 0,Y 495.888,Z 513.522,A -85,B 0,C 180,E1 -6125.693,E2 -6125.693} C_VEL
LIN {X 0,Y 495.864,Z 513.528,A -85,B 0,C 180,E1 -6128.148,E2 -6128.148} C_VEL
LIN {X 0,Y 495.842,Z 513.528,A -85,B 0,C 180,E1 -6131.445,E2 -6131.445} C_VEL
LIN {X 0,Y 495.785,Z 513.541,A -85,B 0,C 180,E1 -6134.783,E2 -6134.783} C_VEL
LIN {X 0,Y 495.779,Z 513.537,A -85,B 0,C 180,E1 -6137.319,E2 -6137.319} C_VEL
LIN {X 0,Y 495.769,Z 513.537,A -85,B 0,C 180,E1 -6139.89,E2 -6139.89} C_VEL
LIN {X 0,Y 495.749,Z 513.546,A -85,B 0,C 180,E1 -6142.861,E2 -6142.861} C_VEL
LIN {X 0,Y 495.791,Z 513.535,A -85,B 0,C 180,E1 -6146.068,E2 -6146.068} C_VEL
LIN {X 0,Y 495.773,Z 513.544,A -85,B 0,C 180,E1 -6148.814,E2 -6148.814} C_VEL
LIN {X 0,Y 495.751,Z 513.539,A -85,B 0,C 180,E1 -6151.726,E2 -6151.726} C_VEL
LIN {X 0,Y 495.77,Z 513.545,A -85,B 0,C 180,E1 -6154.696,E2 -6154.696} C_VEL
LIN {X 0,Y 495.724,Z 513.543,A -85,B 0,C 180,E1 -6157.562,E2 -6157.562} C_VEL
LIN {X 0,Y 495.76,Z 513.545,A -85,B 0,C 180,E1 -6160.7,E2 -6160.7} C_VEL
LIN {X 0,Y 495.728,Z 513.542,A -85,B 0,C 180,E1 -6163.696,E2 -6163.696} C_VEL
LIN {X 0,Y 495.729,Z 513.544,A -85,B 0,C 180,E1 -6166.305,E2 -6166.305} C_VEL
LIN {X 0,Y 495.762,Z 513.541,A -85,B 0,C 180,E1 -6169.301,E2 -6169.301} C_VEL
LIN {X 0,Y 495.727,Z 513.545,A -85,B 0,C 180,E1 -6172.439,E2 -6172.439} C_VEL
LIN {X 0,Y 495.78,Z 513.541,A -85,B 0,C 180,E1 -6175.458,E2 -6175.458} C_VEL
LIN {X 0,Y 495.756,Z 513.545,A -85,B 0,C 180,E1 -6178.365,E2 -6178.365} C_VEL
LIN {X 0,Y 495.819,Z 513.712,A -85,B 0,C 180,E1 -6179.776,E2 -6179.776} C_VEL
LIN {X 0,Y 498.218,Z 525.929,A -85,B 0,C 180,E1 -6182.029,E2 -6182.029} C_VEL
LIN {X 0,Y 497.942,Z 536.65,A -85,B 0,C 180,E1 -6183.829,E2 -6183.829} C_VEL
LIN {X 0,Y 497.321,Z 554.809,A -85,B 0,C 180,E1 -6186.815,E2 -6186.815} C_VEL
LIN {X 0,Y 496.719,Z 574.108,A -85,B 0,C 180,E1 -6189.934,E2 -6189.934} C_VEL
LIN {X 0,Y 496.357,Z 589.007,A -85,B 0,C 180,E1 -6192.277,E2 -6192.277} C_VEL
LIN {X 0,Y 495.969,Z 609.374,A -85,B 0,C 180,E1 -6195.433,E2 -6195.433} C_VEL
LIN {X 0,Y 495.725,Z 621.187,A -85,B 0,C 180,E1 -6197.254,E2 -6197.254} C_VEL
LIN {X 0,Y 497.094,Z 635.465,A -85,B 0,C 180,E1 -6197.531,E2 -6197.531} C_VEL
LIN {X 0,Y 497.201,Z 648.272,A -85,B 0,C 180,E1 -6197.738,E2 -6197.738} C_VEL
LIN {X 0,Y 496.941,Z 701.173,A -85,B 0,C 180,E1 -6198.557,E2 -6198.557} C_VEL
LIN {X 0,Y 496.622,Z 712.78,A -85,B 0,C 180,E1 -6198.883,E2 -6198.883} C_VEL
LIN {X 0,Y 496.395,Z 724.456,A -85,B 0,C 180,E1 -6199.394,E2 -6199.394} C_VEL
LIN {X 0,Y 496.1,Z 734.689,A -85,B 0,C 180,E1 -6200.006,E2 -6200.006} C_VEL
LIN {X 0,Y 495.875,Z 744.027,A -85,B 0,C 180,E1 -6200.723,E2 -6200.723} C_VEL
LIN {X 0,Y 495.576,Z 753.464,A -85,B 0,C 180,E1 -6201.642,E2 -6201.642} C_VEL
LIN {X 0,Y 495.386,Z 761.687,A -85,B 0,C 180,E1 -6202.664,E2 -6202.664} C_VEL
LIN {X 0,Y 495.324,Z 768.269,A -85,B 0,C 180,E1 -6203.689,E2 -6203.689} C_VEL
LIN {X 0,Y 495.173,Z 773.484,A -85,B 0,C 180,E1 -6204.707,E2 -6204.707} C_VEL
LIN {X 0,Y 495.193,Z 778.305,A -85,B 0,C 180,E1 -6205.931,E2 -6205.931} C_VEL
LIN {X 0,Y 495.148,Z 780.691,A -85,B 0,C 180,E1 -6206.745,E2 -6206.745} C_VEL
LIN {X 0,Y 495.119,Z 782.497,A -85,B 0,C 180,E1 -6207.559,E2 -6207.559} C_VEL
LIN {X 0,Y 495.074,Z 783.764,A -85,B 0,C 180,E1 -6208.373,E2 -6208.373} C_VEL
LIN {X 0,Y 495.054,Z 784.537,A -85,B 0,C 180,E1 -6209.187,E2 -6209.187} C_VEL
LIN {X 0,Y 495.118,Z 784.808,A -85,B 0,C 180,E1 -6210,E2 -6210} C_VEL
LIN {X 0,Y 495.058,Z 784.511,A -85,B 0,C 180,E1 -6210.813,E2 -6210.813} C_VEL
LIN {X 0,Y 495.084,Z 783.689,A -85,B 0,C 180,E1 -6211.627,E2 -6211.627} C_VEL
LIN {X 0,Y 495.135,Z 782.371,A -85,B 0,C 180,E1 -6212.44,E2 -6212.44} C_VEL
LIN {X 0,Y 495.202,Z 779.355,A -85,B 0,C 180,E1 -6213.662,E2 -6213.662} C_VEL
LIN {X 0,Y 495.17,Z 774.992,A -85,B 0,C 180,E1 -6214.885,E2 -6214.885} C_VEL
LIN {X 0,Y 495.329,Z 769.064,A -85,B 0,C 180,E1 -6216.108,E2 -6216.108} C_VEL
LIN {X 0,Y 495.371,Z 762.819,A -85,B 0,C 180,E1 -6217.11,E2 -6217.11} C_VEL
LIN {X 0,Y 495.554,Z 754.701,A -85,B 0,C 180,E1 -6218.153,E2 -6218.153} C_VEL
LIN {X 0,Y 495.759,Z 745.646,A -85,B 0,C 180,E1 -6219.074,E2 -6219.074} C_VEL
LIN {X 0,Y 496.043,Z 735.33,A -85,B 0,C 180,E1 -6219.892,E2 -6219.892} C_VEL
LIN {X 0,Y 496.289,Z 725.342,A -85,B 0,C 180,E1 -6220.505,E2 -6220.505} C_VEL
LIN {X 0,Y 496.539,Z 714.214,A -85,B 0,C 180,E1 -6221.015,E2 -6221.015} C_VEL
LIN {X 0,Y 496.822,Z 702.827,A -85,B 0,C 180,E1 -6221.371,E2 -6221.371} C_VEL
LIN {X 0,Y 496.982,Z 683.607,A -85,B 0,C 180,E1 -6221.697,E2 -6221.697} C_VEL
LIN {X 0,Y 497.008,Z 635.007,A -85,B 0,C 180,E1 -6222.424,E2 -6222.424} C_VEL
LIN {X 0,Y 495.703,Z 619.709,A -85,B 0,C 180,E1 -6222.704,E2 -6222.704} C_VEL
LIN {X 0,Y 495.749,Z 616.581,A -85,B 0,C 180,E1 -6223.11,E2 -6223.11} C_VEL
LIN {X 0,Y 495.988,Z 598.58,A -85,B 0,C 180,E1 -6225.829,E2 -6225.829} C_VEL
LIN {X 0,Y 496.327,Z 577.737,A -85,B 0,C 180,E1 -6229.006,E2 -6229.006} C_VEL
LIN {X 0,Y 496.67,Z 559.677,A -85,B 0,C 180,E1 -6231.804,E2 -6231.804} C_VEL
LIN {X 0,Y 497.127,Z 541.717,A -85,B 0,C 180,E1 -6234.648,E2 -6234.648} C_VEL
LIN {X 0,Y 497.549,Z 523.695,A -85,B 0,C 180,E1 -6237.592,E2 -6237.592} C_VEL
LIN {X 0,Y 495.842,Z 513.697,A -85,B 0,C 180,E1 -6239.39,E2 -6239.39} C_VEL
LIN {X 0,Y 495.766,Z 513.544,A -85,B 0,C 180,E1 -6242.594,E2 -6242.594} C_VEL
LIN {X 0,Y 495.751,Z 513.543,A -85,B 0,C 180,E1 -6245.536,E2 -6245.536} C_VEL
LIN {X 0,Y 495.76,Z 513.545,A -85,B 0,C 180,E1 -6248.768,E2 -6248.768} C_VEL
LIN {X 0,Y 495.772,Z 513.538,A -85,B 0,C 180,E1 -6251.778,E2 -6251.778} C_VEL
LIN {X 0,Y 495.743,Z 513.547,A -85,B 0,C 180,E1 -6255.139,E2 -6255.139} C_VEL
LIN {X 0,Y 495.772,Z 513.536,A -85,B 0,C 180,E1 -6258.221,E2 -6258.221} C_VEL
LIN {X 0,Y 495.772,Z 513.542,A -85,B 0,C 180,E1 -6261.229,E2 -6261.229} C_VEL
LIN {X 0,Y 495.751,Z 513.541,A -85,B 0,C 180,E1 -6264.463,E2 -6264.463} C_VEL
LIN {X 0,Y 495.761,Z 513.54,A -85,B 0,C 180,E1 -6267.405,E2 -6267.405} C_VEL
LIN {X 0,Y 495.773,Z 513.538,A -85,B 0,C 180,E1 -6270.254,E2 -6270.254} C_VEL
LIN {X 0,Y 495.825,Z 513.533,A -85,B 0,C 180,E1 -6273.248,E2 -6273.248} C_VEL
LIN {X 0,Y 495.743,Z 513.541,A -85,B 0,C 180,E1 -6275.725,E2 -6275.725} C_VEL
LIN {X 0,Y 495.738,Z 513.544,A -85,B 0,C 180,E1 -6278.371,E2 -6278.371} C_VEL
LIN {X 0,Y 495.776,Z 513.544,A -85,B 0,C 180,E1 -6280.972,E2 -6280.972} C_VEL
LIN {X 0,Y 495.771,Z 513.539,A -85,B 0,C 180,E1 -6283.53,E2 -6283.53} C_VEL
LIN {X 0,Y 495.787,Z 513.537,A -85,B 0,C 180,E1 -6286.056,E2 -6286.056} C_VEL
LIN {X 0,Y 495.865,Z 513.531,A -85,B 0,C 180,E1 -6288.555,E2 -6288.555} C_VEL
LIN {X 0,Y 495.864,Z 513.528,A -85,B 0,C 180,E1 -6291.852,E2 -6291.852} C_VEL
LIN {X 0,Y 495.907,Z 513.524,A -85,B 0,C 180,E1 -6294.307,E2 -6294.307} C_VEL
LIN {X 0,Y 495.985,Z 513.514,A -85,B 0,C 180,E1 -6297.564,E2 -6297.564} C_VEL
LIN {X 0,Y 495.988,Z 513.513,A -85,B 0,C 180,E1 -6300,E2 -6300} C_VEL
LIN {X 0,Y 495.985,Z 513.516,A -85,B 0,C 180,E1 -6302.437,E2 -6302.437} C_VEL
LIN {X 0,Y 495.924,Z 513.667,A -85,B 0,C 180,E1 -6306.28,E2 -6306.28} C_VEL
LIN {X 0,Y 496.049,Z 514.433,A -85,B 0,C 180,E1 -6306.406,E2 -6306.406} C_VEL
LIN {X 0,Y 497.823,Z 520.167,A -85,B 0,C 180,E1 -6306.561,E2 -6306.561} C_VEL
LIN {X 0,Y 497.794,Z 544.751,A -85,B 0,C 180,E1 -6306.944,E2 -6306.944} C_VEL
LIN {X 0,Y 497.776,Z 558.173,A -85,B 0,C 180,E1 -6307.326,E2 -6307.326} C_VEL
LIN {X 0,Y 497.609,Z 569.809,A -85,B 0,C 180,E1 -6307.813,E2 -6307.813} C_VEL
LIN {X 0,Y 497.391,Z 581.62,A -85,B 0,C 180,E1 -6308.485,E2 -6308.485} C_VEL
LIN {X 0,Y 497.142,Z 592.186,A -85,B 0,C 180,E1 -6309.254,E2 -6309.254} C_VEL
LIN {X 0,Y 496.793,Z 602.462,A -85,B 0,C 180,E1 -6310.186,E2 -6310.186} C_VEL
LIN {X 0,Y 496.495,Z 611.606,A -85,B 0,C 180,E1 -6311.224,E2 -6311.224} C_VEL
LIN {X 0,Y 496.222,Z 620.318,A -85,B 0,C 180,E1 -6312.453,E2 -6312.453} C_VEL
LIN {X 0,Y 495.974,Z 627.524,A -85,B 0,C 180,E1 -6313.73,E2 -6313.73} C_VEL
LIN {X 0,Y 495.769,Z 633.505,A -85,B 0,C 180,E1 -6315.096,E2 -6315.096} C_VEL
LIN {X 0,Y 495.565,Z 638.106,A -85,B 0,C 180,E1 -6316.478,E2 -6316.478} C_VEL
LIN {X 0,Y 495.49,Z 640.264,A -85,B 0,C 180,E1 -6317.33,E2 -6317.33} C_VEL
LIN {X 0,Y 495.457,Z 641.926,A -85,B 0,C 180,E1 -6318.184,E2 -6318.184} C_VEL
LIN {X 0,Y 495.401,Z 643.173,A -85,B 0,C 180,E1 -6319.044,E2 -6319.044} C_VEL
LIN {X 0,Y 495.355,Z 644.24,A -85,B 0,C 180,E1 -6320.549,E2 -6320.549} C_VEL
LIN {X 0,Y 495.33,Z 644.182,A -85,B 0,C 180,E1 -6321.648,E2 -6321.648} C_VEL
LIN {X 0,Y 495.359,Z 643.365,A -85,B 0,C 180,E1 -6322.754,E2 -6322.754} C_VEL
LIN {X 0,Y 495.433,Z 641.048,A -85,B 0,C 180,E1 -6324.292,E2 -6324.292} C_VEL
LIN {X 0,Y 495.568,Z 637.777,A -85,B 0,C 180,E1 -6325.629,E2 -6325.629} C_VEL
LIN {X 0,Y 495.721,Z 633.214,A -85,B 0,C 180,E1 -6326.98,E2 -6326.98} C_VEL
LIN {X 0,Y 495.868,Z 627.864,A -85,B 0,C 180,E1 -6328.204,E2 -6328.204} C_VEL
LIN {X 0,Y 496.088,Z 620.788,A -85,B 0,C 180,E1 -6329.492,E2 -6329.492} C_VEL
LIN {X 0,Y 496.391,Z 612.846,A -85,B 0,C 180,E1 -6330.644,E2 -6330.644} C_VEL
LIN {X 0,Y 496.7,Z 603.946,A -85,B 0,C 180,E1 -6331.693,E2 -6331.693} C_VEL
LIN {X 0,Y 496.951,Z 594.24,A -85,B 0,C 180,E1 -6332.628,E2 -6332.628} C_VEL
LIN {X 0,Y 497.285,Z 583.659,A -85,B 0,C 180,E1 -6333.448,E2 -6333.448} C_VEL
LIN {X 0,Y 497.539,Z 572.38,A -85,B 0,C 180,E1 -6334.135,E2 -6334.135} C_VEL
LIN {X 0,Y 497.745,Z 560.263,A -85,B 0,C 180,E1 -6334.695,E2 -6334.695} C_VEL
LIN {X 0,Y 497.873,Z 548.18,A -85,B 0,C 180,E1 -6335.093,E2 -6335.093} C_VEL
LIN {X 0,Y 497.919,Z 534.884,A -85,B 0,C 180,E1 -6335.36,E2 -6335.36} C_VEL
LIN {X 0,Y 497.796,Z 520.189,A -85,B 0,C 180,E1 -6335.581,E2 -6335.581} C_VEL
LIN {X 0,Y 495.954,Z 514.46,A -85,B 0,C 180,E1 -6335.742,E2 -6335.742} C_VEL
LIN {X 0,Y 495.772,Z 513.603,A -85,B 0,C 180,E1 -6335.915,E2 -6335.915} C_VEL
LIN {X 0,Y 495.76,Z 513.544,A -85,B 0,C 180,E1 -6338.773,E2 -6338.773} C_VEL
LIN {X 0,Y 495.774,Z 513.541,A -85,B 0,C 180,E1 -6341.78,E2 -6341.78} C_VEL
LIN {X 0,Y 495.739,Z 513.542,A -85,B 0,C 180,E1 -6342.314,E2 -6342.314} C_VEL
LIN {X 0,Y 495.064,Z 513.631,A -85,B 0,C 180,E1 -6342.992,E2 -6342.992} C_VEL
LIN {X 0,Y 492.197,Z 513.984,A -85,B 0,C 180,E1 -6344.093,E2 -6344.093} C_VEL
LIN {X 0,Y 489.789,Z 514.285,A -85,B 0,C 180,E1 -6344.98,E2 -6344.98} C_VEL
LIN {X 0,Y 488.771,Z 514.413,A -85,B 0,C 180,E1 -6345.666,E2 -6345.666} C_VEL
LIN {X 0,Y 488.697,Z 514.419,A -85,B 0,C 180,E1 -6345.898,E2 -6345.898} C_VEL
LIN {X 0,Y 488.721,Z 514.415,A -85,B 0,C 180,E1 -6348.587,E2 -6348.587} C_VEL
LIN {X 0,Y 488.74,Z 514.415,A -85,B 0,C 180,E1 -6350.943,E2 -6350.943} C_VEL
LIN {X 0,Y 488.676,Z 514.424,A -85,B 0,C 180,E1 -6353.869,E2 -6353.869} C_VEL
LIN {X 0,Y 488.739,Z 514.414,A -85,B 0,C 180,E1 -6356.878,E2 -6356.878} C_VEL
LIN {X 0,Y 488.725,Z 514.419,A -85,B 0,C 180,E1 -6359.782,E2 -6359.782} C_VEL
LIN {X 0,Y 488.794,Z 514.409,A -85,B 0,C 180,E1 -6363.057,E2 -6363.057} C_VEL
LIN {X 0,Y 488.691,Z 514.419,A -85,B 0,C 180,E1 -6366.255,E2 -6366.255} C_VEL
LIN {X 0,Y 488.749,Z 514.415,A -85,B 0,C 180,E1 -6369.176,E2 -6369.176} C_VEL
LIN {X 0,Y 488.753,Z 514.42,A -85,B 0,C 180,E1 -6371.632,E2 -6371.632} C_VEL
LIN {X 0,Y 488.766,Z 514.411,A -85,B 0,C 180,E1 -6375,E2 -6375} C_VEL
LIN {X 0,Y 488.81,Z 514.404,A -85,B 0,C 180,E1 -6378.388,E2 -6378.388} C_VEL
LIN {X 0,Y 488.821,Z 514.411,A -85,B 0,C 180,E1 -6381.734,E2 -6381.734} C_VEL
LIN {X 0,Y 488.81,Z 514.405,A -85,B 0,C 180,E1 -6385.051,E2 -6385.051} C_VEL
LIN {X 0,Y 488.965,Z 514.391,A -85,B 0,C 180,E1 -6387.529,E2 -6387.529} C_VEL
LIN {X 0,Y 488.939,Z 514.388,A -85,B 0,C 180,E1 -6390.824,E2 -6390.824} C_VEL
LIN {X 0,Y 488.966,Z 514.385,A -85,B 0,C 180,E1 -6392.471,E2 -6392.471} C_VEL
LIN {X 0,Y 488.843,Z 514.409,A -85,B 0,C 180,E1 -6395.776,E2 -6395.776} C_VEL
LIN {X 0,Y 488.791,Z 514.409,A -85,B 0,C 180,E1 -6398.267,E2 -6398.267} C_VEL
LIN {X 0,Y 488.811,Z 514.409,A -85,B 0,C 180,E1 -6401.612,E2 -6401.612} C_VEL
LIN {X 0,Y 488.767,Z 514.409,A -85,B 0,C 180,E1 -6405,E2 -6405} C_VEL
LIN {X 0,Y 488.759,Z 514.412,A -85,B 0,C 180,E1 -6408.442,E2 -6408.442} C_VEL
LIN {X 0,Y 488.71,Z 514.416,A -85,B 0,C 180,E1 -6411.07,E2 -6411.07} C_VEL
LIN {X 0,Y 488.683,Z 514.426,A -85,B 0,C 180,E1 -6413.745,E2 -6413.745} C_VEL
LIN {X 0,Y 488.794,Z 514.406,A -85,B 0,C 180,E1 -6416.943,E2 -6416.943} C_VEL
LIN {X 0,Y 488.711,Z 514.42,A -85,B 0,C 180,E1 -6420.362,E2 -6420.362} C_VEL
LIN {X 0,Y 488.735,Z 514.415,A -85,B 0,C 180,E1 -6423.483,E2 -6423.483} C_VEL
LIN {X 0,Y 488.682,Z 514.424,A -85,B 0,C 180,E1 -6426.354,E2 -6426.354} C_VEL
LIN {X 0,Y 488.742,Z 514.413,A -85,B 0,C 180,E1 -6429.249,E2 -6429.249} C_VEL
LIN {X 0,Y 488.73,Z 514.417,A -85,B 0,C 180,E1 -6432.52,E2 -6432.52} C_VEL
LIN {X 0,Y 488.71,Z 514.416,A -85,B 0,C 180,E1 -6435.198,E2 -6435.198} C_VEL
LIN {X 0,Y 488.705,Z 514.422,A -85,B 0,C 180,E1 -6438.399,E2 -6438.399} C_VEL
LIN {X 0,Y 488.701,Z 514.418,A -85,B 0,C 180,E1 -6440.946,E2 -6440.946} C_VEL
LIN {X 0,Y 488.681,Z 514.424,A -85,B 0,C 180,E1 -6443.868,E2 -6443.868} C_VEL
LIN {X 0,Y 488.734,Z 514.414,A -85,B 0,C 180,E1 -6446.876,E2 -6446.876} C_VEL
LIN {X 0,Y 488.729,Z 514.417,A -85,B 0,C 180,E1 -6449.781,E2 -6449.781} C_VEL
LIN {X 0,Y 488.793,Z 514.406,A -85,B 0,C 180,E1 -6453.054,E2 -6453.054} C_VEL
LIN {X 0,Y 488.687,Z 514.428,A -85,B 0,C 180,E1 -6456.254,E2 -6456.254} C_VEL
LIN {X 0,Y 488.739,Z 514.413,A -85,B 0,C 180,E1 -6459.175,E2 -6459.175} C_VEL
LIN {X 0,Y 488.752,Z 514.412,A -85,B 0,C 180,E1 -6461.627,E2 -6461.627} C_VEL
LIN {X 0,Y 488.754,Z 514.412,A -85,B 0,C 180,E1 -6464.999,E2 -6464.999} C_VEL
LIN {X 0,Y 488.821,Z 514.412,A -85,B 0,C 180,E1 -6468.388,E2 -6468.388} C_VEL
LIN {X 0,Y 488.81,Z 514.405,A -85,B 0,C 180,E1 -6471.733,E2 -6471.733} C_VEL
LIN {X 0,Y 488.861,Z 514.403,A -85,B 0,C 180,E1 -6474.224,E2 -6474.224} C_VEL
LIN {X 0,Y 488.953,Z 514.386,A -85,B 0,C 180,E1 -6477.528,E2 -6477.528} C_VEL
LIN {X 0,Y 488.946,Z 514.391,A -85,B 0,C 180,E1 -6480.823,E2 -6480.823} C_VEL
LIN {X 0,Y 488.953,Z 514.395,A -85,B 0,C 180,E1 -6482.471,E2 -6482.471} C_VEL
LIN {X 0,Y 488.847,Z 514.4,A -85,B 0,C 180,E1 -6485.776,E2 -6485.776} C_VEL
LIN {X 0,Y 488.809,Z 514.409,A -85,B 0,C 180,E1 -6488.266,E2 -6488.266} C_VEL
LIN {X 0,Y 488.796,Z 514.406,A -85,B 0,C 180,E1 -6491.612,E2 -6491.612} C_VEL
LIN {X 0,Y 488.755,Z 514.414,A -85,B 0,C 180,E1 -6495,E2 -6495} C_VEL
LIN {X 0,Y 488.746,Z 514.418,A -85,B 0,C 180,E1 -6498.442,E2 -6498.442} C_VEL
LIN {X 0,Y 488.699,Z 514.421,A -85,B 0,C 180,E1 -6501.071,E2 -6501.071} C_VEL
LIN {X 0,Y 488.685,Z 514.419,A -85,B 0,C 180,E1 -6503.746,E2 -6503.746} C_VEL
LIN {X 0,Y 488.791,Z 514.412,A -85,B 0,C 180,E1 -6506.946,E2 -6506.946} C_VEL
LIN {X 0,Y 488.711,Z 514.42,A -85,B 0,C 180,E1 -6510.365,E2 -6510.365} C_VEL
LIN {X 0,Y 488.729,Z 514.415,A -85,B 0,C 180,E1 -6513.485,E2 -6513.485} C_VEL
LIN {X 0,Y 488.682,Z 514.423,A -85,B 0,C 180,E1 -6516.356,E2 -6516.356} C_VEL
LIN {X 0,Y 488.695,Z 514.421,A -85,B 0,C 180,E1 -6519.255,E2 -6519.255} C_VEL
LIN {X 0,Y 488.717,Z 514.416,A -85,B 0,C 180,E1 -6521.602,E2 -6521.602} C_VEL
LIN {X 0,Y 488.706,Z 514.425,A -85,B 0,C 180,E1 -6524.802,E2 -6524.802} C_VEL
LIN {X 0,Y 488.69,Z 514.42,A -85,B 0,C 180,E1 -6527.475,E2 -6527.475} C_VEL
LIN {X 0,Y 488.728,Z 514.414,A -85,B 0,C 180,E1 -6529.677,E2 -6529.677} C_VEL
LIN {X 0,Y 488.678,Z 514.428,A -85,B 0,C 180,E1 -6532.842,E2 -6532.842} C_VEL
LIN {X 0,Y 488.73,Z 514.417,A -85,B 0,C 180,E1 -6535.888,E2 -6535.888} C_VEL
LIN {X 0,Y 488.752,Z 514.448,A -85,B 0,C 180,E1 -6539.488,E2 -6539.488} C_VEL
LIN {X 0,Y 488.996,Z 515.657,A -85,B 0,C 180,E1 -6539.8,E2 -6539.8} C_VEL
LIN {X 0,Y 491.326,Z 527.809,A -85,B 0,C 180,E1 -6542.042,E2 -6542.042} C_VEL
LIN {X 0,Y 490.735,Z 543.975,A -85,B 0,C 180,E1 -6544.783,E2 -6544.783} C_VEL
LIN {X 0,Y 490.133,Z 561.357,A -85,B 0,C 180,E1 -6547.668,E2 -6547.668} C_VEL
LIN {X 0,Y 489.509,Z 582.492,A -85,B 0,C 180,E1 -6551.12,E2 -6551.12} C_VEL
LIN {X 0,Y 488.957,Z 604.99,A -85,B 0,C 180,E1 -6554.68,E2 -6554.68} C_VEL
LIN {X 0,Y 488.641,Z 619.977,A -85,B 0,C 180,E1 -6557.039,E2 -6557.039} C_VEL
LIN {X 0,Y 489.284,Z 627.111,A -85,B 0,C 180,E1 -6557.195,E2 -6557.195} C_VEL
LIN {X 0,Y 490.341,Z 638.773,A -85,B 0,C 180,E1 -6557.411,E2 -6557.411} C_VEL
LIN {X 0,Y 489.951,Z 700.494,A -85,B 0,C 180,E1 -6558.392,E2 -6558.392} C_VEL
LIN {X 0,Y 489.601,Z 713.252,A -85,B 0,C 180,E1 -6558.774,E2 -6558.774} C_VEL
LIN {X 0,Y 489.402,Z 723.506,A -85,B 0,C 180,E1 -6559.241,E2 -6559.241} C_VEL
LIN {X 0,Y 489.078,Z 733.734,A -85,B 0,C 180,E1 -6559.862,E2 -6559.862} C_VEL
LIN {X 0,Y 488.797,Z 744.227,A -85,B 0,C 180,E1 -6560.691,E2 -6560.691} C_VEL
LIN {X 0,Y 488.505,Z 752.474,A -85,B 0,C 180,E1 -6561.52,E2 -6561.52} C_VEL
LIN {X 0,Y 488.314,Z 760.713,A -85,B 0,C 180,E1 -6562.558,E2 -6562.558} C_VEL
LIN {X 0,Y 488.242,Z 767.126,A -85,B 0,C 180,E1 -6563.567,E2 -6563.567} C_VEL
LIN {X 0,Y 488.119,Z 772.506,A -85,B 0,C 180,E1 -6564.63,E2 -6564.63} C_VEL
LIN {X 0,Y 488.129,Z 777.326,A -85,B 0,C 180,E1 -6565.872,E2 -6565.872} C_VEL
LIN {X 0,Y 488.103,Z 779.714,A -85,B 0,C 180,E1 -6566.698,E2 -6566.698} C_VEL
LIN {X 0,Y 488.071,Z 781.53,A -85,B 0,C 180,E1 -6567.524,E2 -6567.524} C_VEL
LIN {X 0,Y 488.035,Z 782.795,A -85,B 0,C 180,E1 -6568.35,E2 -6568.35} C_VEL
LIN {X 0,Y 488.02,Z 783.555,A -85,B 0,C 180,E1 -6569.175,E2 -6569.175} C_VEL
LIN {X 0,Y 488.103,Z 783.821,A -85,B 0,C 180,E1 -6570,E2 -6570} C_VEL
LIN {X 0,Y 488.025,Z 783.513,A -85,B 0,C 180,E1 -6570.825,E2 -6570.825} C_VEL
LIN {X 0,Y 488.048,Z 782.694,A -85,B 0,C 180,E1 -6571.65,E2 -6571.65} C_VEL
LIN {X 0,Y 488.092,Z 781.361,A -85,B 0,C 180,E1 -6572.476,E2 -6572.476} C_VEL
LIN {X 0,Y 488.156,Z 778.329,A -85,B 0,C 180,E1 -6573.714,E2 -6573.714} C_VEL
LIN {X 0,Y 488.127,Z 773.929,A -85,B 0,C 180,E1 -6574.956,E2 -6574.956} C_VEL
LIN {X 0,Y 488.262,Z 767.976,A -85,B 0,C 180,E1 -6576.197,E2 -6576.197} C_VEL
LIN {X 0,Y 488.305,Z 761.712,A -85,B 0,C 180,E1 -6577.214,E2 -6577.214} C_VEL
LIN {X 0,Y 488.482,Z 753.575,A -85,B 0,C 180,E1 -6578.272,E2 -6578.272} C_VEL
LIN {X 0,Y 488.748,Z 744.486,A -85,B 0,C 180,E1 -6579.205,E2 -6579.205} C_VEL
LIN {X 0,Y 489.022,Z 734.147,A -85,B 0,C 180,E1 -6580.035,E2 -6580.035} C_VEL
LIN {X 0,Y 489.26,Z 724.165,A -85,B 0,C 180,E1 -6580.658,E2 -6580.658} C_VEL
LIN {X 0,Y 489.537,Z 713.007,A -85,B 0,C 180,E1 -6581.175,E2 -6581.175} C_VEL
LIN {X 0,Y 489.882,Z 701.667,A -85,B 0,C 180,E1 -6581.534,E2 -6581.534} C_VEL
LIN {X 0,Y 490.017,Z 683.212,A -85,B 0,C 180,E1 -6581.855,E2 -6581.855} C_VEL
LIN {X 0,Y 490.046,Z 635.492,A -85,B 0,C 180,E1 -6582.589,E2 -6582.589} C_VEL
LIN {X 0,Y 488.648,Z 618.223,A -85,B 0,C 180,E1 -6582.907,E2 -6582.907} C_VEL
LIN {X 0,Y 488.657,Z 616.529,A -85,B 0,C 180,E1 -6583.092,E2 -6583.092} C_VEL
LIN {X 0,Y 488.902,Z 598.587,A -85,B 0,C 180,E1 -6585.85,E2 -6585.85} C_VEL
LIN {X 0,Y 489.224,Z 579.479,A -85,B 0,C 180,E1 -6588.814,E2 -6588.814} C_VEL
LIN {X 0,Y 489.62,Z 561.229,A -85,B 0,C 180,E1 -6591.691,E2 -6591.691} C_VEL
LIN {X 0,Y 490.064,Z 543.345,A -85,B 0,C 180,E1 -6594.575,E2 -6594.575} C_VEL
LIN {X 0,Y 490.568,Z 525.65,A -85,B 0,C 180,E1 -6597.516,E2 -6597.516} C_VEL
LIN {X 0,Y 489.766,Z 519.84,A -85,B 0,C 180,E1 -6598.545,E2 -6598.545} C_VEL
LIN {X 0,Y 488.773,Z 514.459,A -85,B 0,C 180,E1 -6599.591,E2 -6599.591} C_VEL
LIN {X 0,Y 488.735,Z 514.42,A -85,B 0,C 180,E1 -6603.122,E2 -6603.122} C_VEL
LIN {X 0,Y 488.679,Z 514.423,A -85,B 0,C 180,E1 -6606.131,E2 -6606.131} C_VEL
LIN {X 0,Y 488.697,Z 514.424,A -85,B 0,C 180,E1 -6609.253,E2 -6609.253} C_VEL
LIN {X 0,Y 488.718,Z 514.417,A -85,B 0,C 180,E1 -6611.601,E2 -6611.601} C_VEL
LIN {X 0,Y 488.706,Z 514.423,A -85,B 0,C 180,E1 -6614.801,E2 -6614.801} C_VEL
LIN {X 0,Y 488.729,Z 514.414,A -85,B 0,C 180,E1 -6617.479,E2 -6617.479} C_VEL
LIN {X 0,Y 488.742,Z 514.419,A -85,B 0,C 180,E1 -6620.75,E2 -6620.75} C_VEL
LIN {X 0,Y 488.679,Z 514.419,A -85,B 0,C 180,E1 -6623.868,E2 -6623.868} C_VEL
LIN {X 0,Y 488.731,Z 514.42,A -85,B 0,C 180,E1 -6626.877,E2 -6626.877} C_VEL
LIN {X 0,Y 488.726,Z 514.415,A -85,B 0,C 180,E1 -6629.781,E2 -6629.781} C_VEL
LIN {X 0,Y 488.79,Z 514.411,A -85,B 0,C 180,E1 -6633.054,E2 -6633.054} C_VEL
LIN {X 0,Y 488.684,Z 514.422,A -85,B 0,C 180,E1 -6636.254,E2 -6636.254} C_VEL
LIN {X 0,Y 488.736,Z 514.417,A -85,B 0,C 180,E1 -6639.175,E2 -6639.175} C_VEL
LIN {X 0,Y 488.749,Z 514.412,A -85,B 0,C 180,E1 -6641.628,E2 -6641.628} C_VEL
LIN {X 0,Y 488.752,Z 514.418,A -85,B 0,C 180,E1 -6645,E2 -6645} C_VEL
LIN {X 0,Y 488.823,Z 514.407,A -85,B 0,C 180,E1 -6648.388,E2 -6648.388} C_VEL
LIN {X 0,Y 488.809,Z 514.407,A -85,B 0,C 180,E1 -6651.734,E2 -6651.734} C_VEL
LIN {X 0,Y 488.864,Z 514.401,A -85,B 0,C 180,E1 -6654.225,E2 -6654.225} C_VEL
LIN {X 0,Y 488.953,Z 514.39,A -85,B 0,C 180,E1 -6657.529,E2 -6657.529} C_VEL
LIN {X 0,Y 488.959,Z 514.389,A -85,B 0,C 180,E1 -6660,E2 -6660} C_VEL
LIN {X 0,Y 488.953,Z 514.392,A -85,B 0,C 180,E1 -6662.472,E2 -6662.472} C_VEL
LIN {X 0,Y 488.888,Z 514.544,A -85,B 0,C 180,E1 -6666.086,E2 -6666.086} C_VEL
LIN {X 0,Y 489.018,Z 515.308,A -85,B 0,C 180,E1 -6666.214,E2 -6666.214} C_VEL
LIN {X 0,Y 490.981,Z 522.142,A -85,B 0,C 180,E1 -6666.395,E2 -6666.395} C_VEL
LIN {X 0,Y 490.926,Z 546.451,A -85,B 0,C 180,E1 -6666.783,E2 -6666.783} C_VEL
LIN {X 0,Y 490.878,Z 559.747,A -85,B 0,C 180,E1 -6667.171,E2 -6667.171} C_VEL
LIN {X 0,Y 490.739,Z 571.229,A -85,B 0,C 180,E1 -6667.665,E2 -6667.665} C_VEL
LIN {X 0,Y 490.489,Z 583.166,A -85,B 0,C 180,E1 -6668.357,E2 -6668.357} C_VEL
LIN {X 0,Y 490.208,Z 594.166,A -85,B 0,C 180,E1 -6669.178,E2 -6669.178} C_VEL
LIN {X 0,Y 489.857,Z 604.244,A -85,B 0,C 180,E1 -6670.123,E2 -6670.123} C_VEL
LIN {X 0,Y 489.551,Z 613.26,A -85,B 0,C 180,E1 -6671.175,E2 -6671.175} C_VEL
LIN {X 0,Y 489.231,Z 622.026,A -85,B 0,C 180,E1 -6672.444,E2 -6672.444} C_VEL
LIN {X 0,Y 488.991,Z 628.963,A -85,B 0,C 180,E1 -6673.718,E2 -6673.718} C_VEL
LIN {X 0,Y 488.778,Z 634.478,A -85,B 0,C 180,E1 -6675,E2 -6675} C_VEL
LIN {X 0,Y 488.585,Z 638.767,A -85,B 0,C 180,E1 -6676.29,E2 -6676.29} C_VEL
LIN {X 0,Y 488.455,Z 641.926,A -85,B 0,C 180,E1 -6677.587,E2 -6677.587} C_VEL
LIN {X 0,Y 488.434,Z 643.457,A -85,B 0,C 180,E1 -6678.455,E2 -6678.455} C_VEL
LIN {X 0,Y 488.368,Z 644.505,A -85,B 0,C 180,E1 -6679.329,E2 -6679.329} C_VEL
LIN {X 0,Y 488.317,Z 645.272,A -85,B 0,C 180,E1 -6680.695,E2 -6680.695} C_VEL
LIN {X 0,Y 488.326,Z 645.008,A -85,B 0,C 180,E1 -6681.975,E2 -6681.975} C_VEL
LIN {X 0,Y 488.339,Z 644.216,A -85,B 0,C 180,E1 -6682.921,E2 -6682.921} C_VEL
LIN {X 0,Y 488.382,Z 643.055,A -85,B 0,C 180,E1 -6683.762,E2 -6683.762} C_VEL
LIN {X 0,Y 488.522,Z 640.564,A -85,B 0,C 180,E1 -6685,E2 -6685} C_VEL
LIN {X 0,Y 488.631,Z 636.27,A -85,B 0,C 180,E1 -6686.48,E2 -6686.48} C_VEL
LIN {X 0,Y 488.787,Z 630.874,A -85,B 0,C 180,E1 -6687.86,E2 -6687.86} C_VEL
LIN {X 0,Y 488.979,Z 625.48,A -85,B 0,C 180,E1 -6688.95,E2 -6688.95} C_VEL
LIN {X 0,Y 489.285,Z 617.992,A -85,B 0,C 180,E1 -6690.181,E2 -6690.181} C_VEL
LIN {X 0,Y 489.589,Z 609.06,A -85,B 0,C 180,E1 -6691.357,E2 -6691.357} C_VEL
LIN {X 0,Y 489.91,Z 599.481,A -85,B 0,C 180,E1 -6692.38,E2 -6692.38} C_VEL
LIN {X 0,Y 490.256,Z 589.49,A -85,B 0,C 180,E1 -6693.243,E2 -6693.243} C_VEL
LIN {X 0,Y 490.584,Z 577.994,A -85,B 0,C 180,E1 -6694.029,E2 -6694.029} C_VEL
LIN {X 0,Y 490.809,Z 565.289,A -85,B 0,C 180,E1 -6694.694,E2 -6694.694} C_VEL
LIN {X 0,Y 490.918,Z 552.518,A -85,B 0,C 180,E1 -6695.171,E2 -6695.171} C_VEL
LIN {X 0,Y 490.989,Z 539.198,A -85,B 0,C 180,E1 -6695.483,E2 -6695.483} C_VEL
LIN {X 0,Y 490.956,Z 521.742,A -85,B 0,C 180,E1 -6695.751,E2 -6695.751} C_VEL
LIN {X 0,Y 488.923,Z 515.4,A -85,B 0,C 180,E1 -6695.928,E2 -6695.928} C_VEL
LIN {X 0,Y 488.719,Z 514.506,A -85,B 0,C 180,E1 -6696.092,E2 -6696.092} C_VEL
LIN {X 0,Y 488.697,Z 514.426,A -85,B 0,C 180,E1 -6699.255,E2 -6699.255} C_VEL
LIN {X 0,Y 488.687,Z 514.421,A -85,B 0,C 180,E1 -6702.314,E2 -6702.314} C_VEL
LIN {X 0,Y 488.709,Z 514.423,A -85,B 0,C 180,E1 -6705.2,E2 -6705.2} C_VEL
LIN {X 0,Y 488.697,Z 514.419,A -85,B 0,C 180,E1 -6705.898,E2 -6705.898} C_VEL
LIN {X 0,Y 488.055,Z 514.501,A -85,B 0,C 180,E1 -6706.586,E2 -6706.586} C_VEL
LIN {X 0,Y 485.218,Z 514.862,A -85,B 0,C 180,E1 -6707.703,E2 -6707.703} C_VEL
LIN {X 0,Y 482.804,Z 515.164,A -85,B 0,C 180,E1 -6708.604,E2 -6708.604} C_VEL
LIN {X 0,Y 481.763,Z 515.29,A -85,B 0,C 180,E1 -6709.299,E2 -6709.299} C_VEL
LIN {X 0,Y 481.678,Z 515.298,A -85,B 0,C 180,E1 -6709.535,E2 -6709.535} C_VEL
LIN {X 0,Y 481.631,Z 515.299,A -85,B 0,C 180,E1 -6712.204,E2 -6712.204} C_VEL
LIN {X 0,Y 481.688,Z 515.298,A -85,B 0,C 180,E1 -6715.319,E2 -6715.319} C_VEL
LIN {X 0,Y 481.646,Z 515.297,A -85,B 0,C 180,E1 -6718.313,E2 -6718.313} C_VEL
LIN {X 0,Y 481.702,Z 515.294,A -85,B 0,C 180,E1 -6721.219,E2 -6721.219} C_VEL
LIN {X 0,Y 481.703,Z 515.291,A -85,B 0,C 180,E1 -6724.044,E2 -6724.044} C_VEL
LIN {X 0,Y 481.677,Z 515.293,A -85,B 0,C 180,E1 -6726.813,E2 -6726.813} C_VEL
LIN {X 0,Y 481.698,Z 515.298,A -85,B 0,C 180,E1 -6729.503,E2 -6729.503} C_VEL
LIN {X 0,Y 481.695,Z 515.292,A -85,B 0,C 180,E1 -6732.159,E2 -6732.159} C_VEL
LIN {X 0,Y 481.747,Z 515.284,A -85,B 0,C 180,E1 -6734.776,E2 -6734.776} C_VEL
LIN {X 0,Y 481.755,Z 515.284,A -85,B 0,C 180,E1 -6738.216,E2 -6738.216} C_VEL
LIN {X 0,Y 481.766,Z 515.289,A -85,B 0,C 180,E1 -6741.612,E2 -6741.612} C_VEL
LIN {X 0,Y 481.78,Z 515.28,A -85,B 0,C 180,E1 -6744.979,E2 -6744.979} C_VEL
LIN {X 0,Y 481.932,Z 515.266,A -85,B 0,C 180,E1 -6747.493,E2 -6747.493} C_VEL
LIN {X 0,Y 481.891,Z 515.266,A -85,B 0,C 180,E1 -6750.836,E2 -6750.836} C_VEL
LIN {X 0,Y 481.932,Z 515.261,A -85,B 0,C 180,E1 -6752.507,E2 -6752.507} C_VEL
LIN {X 0,Y 481.802,Z 515.285,A -85,B 0,C 180,E1 -6755.861,E2 -6755.861} C_VEL
LIN {X 0,Y 481.746,Z 515.286,A -85,B 0,C 180,E1 -6758.388,E2 -6758.388} C_VEL
LIN {X 0,Y 481.756,Z 515.291,A -85,B 0,C 180,E1 -6761.785,E2 -6761.785} C_VEL
LIN {X 0,Y 481.747,Z 515.285,A -85,B 0,C 180,E1 -6765.224,E2 -6765.224} C_VEL
LIN {X 0,Y 481.716,Z 515.288,A -85,B 0,C 180,E1 -6768.721,E2 -6768.721} C_VEL
LIN {X 0,Y 481.649,Z 515.298,A -85,B 0,C 180,E1 -6771.394,E2 -6771.394} C_VEL
LIN {X 0,Y 481.664,Z 515.3,A -85,B 0,C 180,E1 -6774.113,E2 -6774.113} C_VEL
LIN {X 0,Y 481.749,Z 515.284,A -85,B 0,C 180,E1 -6777.139,E2 -6777.139} C_VEL
LIN {X 0,Y 481.68,Z 515.297,A -85,B 0,C 180,E1 -6779.74,E2 -6779.74} C_VEL
LIN {X 0,Y 481.673,Z 515.294,A -85,B 0,C 180,E1 -6782.673,E2 -6782.673} C_VEL
LIN {X 0,Y 481.636,Z 515.302,A -85,B 0,C 180,E1 -6785.709,E2 -6785.709} C_VEL
LIN {X 0,Y 481.714,Z 515.289,A -85,B 0,C 180,E1 -6789.353,E2 -6789.353} C_VEL
LIN {X 0,Y 481.672,Z 515.301,A -85,B 0,C 180,E1 -6792.157,E2 -6792.157} C_VEL
LIN {X 0,Y 481.658,Z 515.299,A -85,B 0,C 180,E1 -6794.456,E2 -6794.456} C_VEL
LIN {X 0,Y 481.645,Z 515.301,A -85,B 0,C 180,E1 -6797.838,E2 -6797.838} C_VEL
LIN {X 0,Y 481.677,Z 515.295,A -85,B 0,C 180,E1 -6800.65,E2 -6800.65} C_VEL
LIN {X 0,Y 481.627,Z 515.299,A -85,B 0,C 180,E1 -6803.375,E2 -6803.375} C_VEL
LIN {X 0,Y 481.705,Z 515.296,A -85,B 0,C 180,E1 -6806.329,E2 -6806.329} C_VEL
LIN {X 0,Y 481.653,Z 515.296,A -85,B 0,C 180,E1 -6809.415,E2 -6809.415} C_VEL
LIN {X 0,Y 481.697,Z 515.298,A -85,B 0,C 180,E1 -6812.167,E2 -6812.167} C_VEL
LIN {X 0,Y 481.712,Z 515.289,A -85,B 0,C 180,E1 -6814.969,E2 -6814.969} C_VEL
LIN {X 0,Y 481.643,Z 515.298,A -85,B 0,C 180,E1 -6817.704,E2 -6817.704} C_VEL
LIN {X 0,Y 481.701,Z 515.297,A -85,B 0,C 180,E1 -6820.392,E2 -6820.392} C_VEL
LIN {X 0,Y 481.684,Z 515.292,A -85,B 0,C 180,E1 -6823.033,E2 -6823.033} C_VEL
LIN {X 0,Y 481.681,Z 515.293,A -85,B 0,C 180,E1 -6825.638,E2 -6825.638} C_VEL
LIN {X 0,Y 481.786,Z 515.285,A -85,B 0,C 180,E1 -6828.216,E2 -6828.216} C_VEL
LIN {X 0,Y 481.755,Z 515.283,A -85,B 0,C 180,E1 -6831.611,E2 -6831.611} C_VEL
LIN {X 0,Y 481.82,Z 515.279,A -85,B 0,C 180,E1 -6834.139,E2 -6834.139} C_VEL
LIN {X 0,Y 481.92,Z 515.262,A -85,B 0,C 180,E1 -6837.492,E2 -6837.492} C_VEL
LIN {X 0,Y 481.897,Z 515.269,A -85,B 0,C 180,E1 -6840.835,E2 -6840.835} C_VEL
LIN {X 0,Y 481.92,Z 515.271,A -85,B 0,C 180,E1 -6842.507,E2 -6842.507} C_VEL
LIN {X 0,Y 481.808,Z 515.277,A -85,B 0,C 180,E1 -6845.86,E2 -6845.86} C_VEL
LIN {X 0,Y 481.754,Z 515.289,A -85,B 0,C 180,E1 -6848.388,E2 -6848.388} C_VEL
LIN {X 0,Y 481.741,Z 515.285,A -85,B 0,C 180,E1 -6851.785,E2 -6851.785} C_VEL
LIN {X 0,Y 481.735,Z 515.287,A -85,B 0,C 180,E1 -6855.224,E2 -6855.224} C_VEL
LIN {X 0,Y 481.703,Z 515.297,A -85,B 0,C 180,E1 -6858.722,E2 -6858.722} C_VEL
LIN {X 0,Y 481.638,Z 515.298,A -85,B 0,C 180,E1 -6861.395,E2 -6861.395} C_VEL
LIN {X 0,Y 481.668,Z 515.295,A -85,B 0,C 180,E1 -6864.113,E2 -6864.113} C_VEL
LIN {X 0,Y 481.744,Z 515.287,A -85,B 0,C 180,E1 -6867.141,E2 -6867.141} C_VEL
LIN {X 0,Y 481.68,Z 515.292,A -85,B 0,C 180,E1 -6869.741,E2 -6869.741} C_VEL
LIN {X 0,Y 481.666,Z 515.302,A -85,B 0,C 180,E1 -6872.674,E2 -6872.674} C_VEL
LIN {X 0,Y 481.636,Z 515.298,A -85,B 0,C 180,E1 -6875.709,E2 -6875.709} C_VEL
LIN {X 0,Y 481.665,Z 515.302,A -85,B 0,C 180,E1 -6878.859,E2 -6878.859} C_VEL
LIN {X 0,Y 481.656,Z 515.295,A -85,B 0,C 180,E1 -6881.915,E2 -6881.915} C_VEL
LIN {X 0,Y 481.654,Z 515.299,A -85,B 0,C 180,E1 -6884.458,E2 -6884.458} C_VEL
LIN {X 0,Y 481.649,Z 515.296,A -85,B 0,C 180,E1 -6887.841,E2 -6887.841} C_VEL
LIN {X 0,Y 481.687,Z 515.297,A -85,B 0,C 180,E1 -6891.143,E2 -6891.143} C_VEL
LIN {X 0,Y 481.663,Z 515.303,A -85,B 0,C 180,E1 -6894.795,E2 -6894.795} C_VEL
LIN {X 0,Y 481.67,Z 515.302,A -85,B 0,C 180,E1 -6897.326,E2 -6897.326} C_VEL
LIN {X 0,Y 481.7,Z 515.435,A -85,B 0,C 180,E1 -6899.344,E2 -6899.344} C_VEL
LIN {X 0,Y 484.345,Z 528.607,A -85,B 0,C 180,E1 -6901.864,E2 -6901.864} C_VEL
LIN {X 0,Y 483.998,Z 539.253,A -85,B 0,C 180,E1 -6903.713,E2 -6903.713} C_VEL
LIN {X 0,Y 483.269,Z 557.919,A -85,B 0,C 180,E1 -6906.881,E2 -6906.881} C_VEL
LIN {X 0,Y 482.525,Z 579.257,A -85,B 0,C 180,E1 -6910.428,E2 -6910.428} C_VEL
LIN {X 0,Y 481.991,Z 596.652,A -85,B 0,C 180,E1 -6913.263,E2 -6913.263} C_VEL
LIN {X 0,Y 481.676,Z 612.655,A -85,B 0,C 180,E1 -6915.854,E2 -6915.854} C_VEL
LIN {X 0,Y 481.58,Z 618.892,A -85,B 0,C 180,E1 -6916.828,E2 -6916.828} C_VEL
LIN {X 0,Y 483.409,Z 638.986,A -85,B 0,C 180,E1 -6917.233,E2 -6917.233} C_VEL
LIN {X 0,Y 483.01,Z 699.727,A -85,B 0,C 180,E1 -6918.224,E2 -6918.224} C_VEL
LIN {X 0,Y 482.664,Z 710.982,A -85,B 0,C 180,E1 -6918.557,E2 -6918.557} C_VEL
LIN {X 0,Y 482.411,Z 722.556,A -85,B 0,C 180,E1 -6919.083,E2 -6919.083} C_VEL
LIN {X 0,Y 482.028,Z 732.776,A -85,B 0,C 180,E1 -6919.712,E2 -6919.712} C_VEL
LIN {X 0,Y 481.702,Z 743.234,A -85,B 0,C 180,E1 -6920.553,E2 -6920.553} C_VEL
LIN {X 0,Y 481.443,Z 751.486,A -85,B 0,C 180,E1 -6921.395,E2 -6921.395} C_VEL
LIN {X 0,Y 481.246,Z 759.74,A -85,B 0,C 180,E1 -6922.448,E2 -6922.448} C_VEL
LIN {X 0,Y 481.154,Z 766.771,A -85,B 0,C 180,E1 -6923.585,E2 -6923.585} C_VEL
LIN {X 0,Y 481.066,Z 771.527,A -85,B 0,C 180,E1 -6924.551,E2 -6924.551} C_VEL
LIN {X 0,Y 481.068,Z 776.348,A -85,B 0,C 180,E1 -6925.811,E2 -6925.811} C_VEL
LIN {X 0,Y 481.059,Z 778.737,A -85,B 0,C 180,E1 -6926.65,E2 -6926.65} C_VEL
LIN {X 0,Y 481.023,Z 780.561,A -85,B 0,C 180,E1 -6927.488,E2 -6927.488} C_VEL
LIN {X 0,Y 480.994,Z 781.825,A -85,B 0,C 180,E1 -6928.325,E2 -6928.325} C_VEL
LIN {X 0,Y 480.986,Z 782.573,A -85,B 0,C 180,E1 -6929.163,E2 -6929.163} C_VEL
LIN {X 0,Y 481.088,Z 782.834,A -85,B 0,C 180,E1 -6930,E2 -6930} C_VEL
LIN {X 0,Y 480.993,Z 782.513,A -85,B 0,C 180,E1 -6930.837,E2 -6930.837} C_VEL
LIN {X 0,Y 481.011,Z 781.699,A -85,B 0,C 180,E1 -6931.674,E2 -6931.674} C_VEL
LIN {X 0,Y 481.048,Z 780.349,A -85,B 0,C 180,E1 -6932.512,E2 -6932.512} C_VEL
LIN {X 0,Y 481.108,Z 777.304,A -85,B 0,C 180,E1 -6933.769,E2 -6933.769} C_VEL
LIN {X 0,Y 481.083,Z 772.866,A -85,B 0,C 180,E1 -6935.028,E2 -6935.028} C_VEL
LIN {X 0,Y 481.19,Z 767.663,A -85,B 0,C 180,E1 -6936.147,E2 -6936.147} C_VEL
LIN {X 0,Y 481.224,Z 760.458,A -85,B 0,C 180,E1 -6937.342,E2 -6937.342} C_VEL
LIN {X 0,Y 481.403,Z 752.433,A -85,B 0,C 180,E1 -6938.394,E2 -6938.394} C_VEL
LIN {X 0,Y 481.725,Z 743.323,A -85,B 0,C 180,E1 -6939.34,E2 -6939.34} C_VEL
LIN {X 0,Y 481.983,Z 732.961,A -85,B 0,C 180,E1 -6940.183,E2 -6940.183} C_VEL
LIN {X 0,Y 482.287,Z 722.006,A -85,B 0,C 180,E1 -6940.867,E2 -6940.867} C_VEL
LIN {X 0,Y 482.63,Z 710.5,A -85,B 0,C 180,E1 -6941.39,E2 -6941.39} C_VEL
LIN {X 0,Y 482.94,Z 698.263,A -85,B 0,C 180,E1 -6941.755,E2 -6941.755} C_VEL
LIN {X 0,Y 483.165,Z 636.594,A -85,B 0,C 180,E1 -6942.746,E2 -6942.746} C_VEL
LIN {X 0,Y 481.567,Z 616.552,A -85,B 0,C 180,E1 -6943.127,E2 -6943.127} C_VEL
LIN {X 0,Y 481.585,Z 613.732,A -85,B 0,C 180,E1 -6943.503,E2 -6943.503} C_VEL
LIN {X 0,Y 481.836,Z 595.823,A -85,B 0,C 180,E1 -6946.306,E2 -6946.306} C_VEL
LIN {X 0,Y 482.217,Z 576.528,A -85,B 0,C 180,E1 -6949.363,E2 -6949.363} C_VEL
LIN {X 0,Y 482.613,Z 558.645,A -85,B 0,C 180,E1 -6952.248,E2 -6952.248} C_VEL
LIN {X 0,Y 483.141,Z 540.311,A -85,B 0,C 180,E1 -6955.278,E2 -6955.278} C_VEL
LIN {X 0,Y 483.568,Z 526.011,A -85,B 0,C 180,E1 -6957.714,E2 -6957.714} C_VEL
LIN {X 0,Y 481.79,Z 515.643,A -85,B 0,C 180,E1 -6959.638,E2 -6959.638} C_VEL
LIN {X 0,Y 481.683,Z 515.3,A -85,B 0,C 180,E1 -6959.981,E2 -6959.981} C_VEL
LIN {X 0,Y 481.706,Z 515.294,A -85,B 0,C 180,E1 -6963.669,E2 -6963.669} C_VEL
LIN {X 0,Y 481.624,Z 515.307,A -85,B 0,C 180,E1 -6966.746,E2 -6966.746} C_VEL
LIN {X 0,Y 481.672,Z 515.294,A -85,B 0,C 180,E1 -6969.94,E2 -6969.94} C_VEL
LIN {X 0,Y 481.675,Z 515.298,A -85,B 0,C 180,E1 -6973.294,E2 -6973.294} C_VEL
LIN {X 0,Y 481.683,Z 515.3,A -85,B 0,C 180,E1 -6976.845,E2 -6976.845} C_VEL
LIN {X 0,Y 481.685,Z 515.293,A -85,B 0,C 180,E1 -6980.061,E2 -6980.061} C_VEL
LIN {X 0,Y 481.624,Z 515.302,A -85,B 0,C 180,E1 -6983.253,E2 -6983.253} C_VEL
LIN {X 0,Y 481.701,Z 515.293,A -85,B 0,C 180,E1 -6986.33,E2 -6986.33} C_VEL
LIN {X 0,Y 481.656,Z 515.298,A -85,B 0,C 180,E1 -6989.414,E2 -6989.414} C_VEL
LIN {X 0,Y 481.694,Z 515.293,A -85,B 0,C 180,E1 -6992.168,E2 -6992.168} C_VEL
LIN {X 0,Y 481.71,Z 515.297,A -85,B 0,C 180,E1 -6994.97,E2 -6994.97} C_VEL
LIN {X 0,Y 481.64,Z 515.299,A -85,B 0,C 180,E1 -6997.705,E2 -6997.705} C_VEL
LIN {X 0,Y 481.699,Z 515.292,A -85,B 0,C 180,E1 -7000.393,E2 -7000.393} C_VEL
LIN {X 0,Y 481.682,Z 515.3,A -85,B 0,C 180,E1 -7003.034,E2 -7003.034} C_VEL
LIN {X 0,Y 481.681,Z 515.294,A -85,B 0,C 180,E1 -7005.639,E2 -7005.639} C_VEL
LIN {X 0,Y 481.786,Z 515.282,A -85,B 0,C 180,E1 -7008.216,E2 -7008.216} C_VEL
LIN {X 0,Y 481.754,Z 515.286,A -85,B 0,C 180,E1 -7011.612,E2 -7011.612} C_VEL
LIN {X 0,Y 481.822,Z 515.278,A -85,B 0,C 180,E1 -7014.14,E2 -7014.14} C_VEL
LIN {X 0,Y 481.92,Z 515.266,A -85,B 0,C 180,E1 -7017.493,E2 -7017.493} C_VEL
LIN {X 0,Y 481.93,Z 515.265,A -85,B 0,C 180,E1 -7020,E2 -7020} C_VEL
LIN {X 0,Y 481.92,Z 515.268,A -85,B 0,C 180,E1 -7022.508,E2 -7022.508} C_VEL
LIN {X 0,Y 481.84,Z 515.439,A -85,B 0,C 180,E1 -7025.887,E2 -7025.887} C_VEL
LIN {X 0,Y 482.059,Z 516.473,A -85,B 0,C 180,E1 -7026.028,E2 -7026.028} C_VEL
LIN {X 0,Y 484.029,Z 522.696,A -85,B 0,C 180,E1 -7026.2,E2 -7026.2} C_VEL
LIN {X 0,Y 484.052,Z 547.187,A -85,B 0,C 180,E1 -7026.592,E2 -7026.592} C_VEL
LIN {X 0,Y 484.017,Z 560.597,A -85,B 0,C 180,E1 -7026.985,E2 -7026.985} C_VEL
LIN {X 0,Y 483.886,Z 571.628,A -85,B 0,C 180,E1 -7027.459,E2 -7027.459} C_VEL
LIN {X 0,Y 483.632,Z 583.527,A -85,B 0,C 180,E1 -7028.146,E2 -7028.146} C_VEL
LIN {X 0,Y 483.324,Z 594.824,A -85,B 0,C 180,E1 -7028.991,E2 -7028.991} C_VEL
LIN {X 0,Y 482.98,Z 605.026,A -85,B 0,C 180,E1 -7029.951,E2 -7029.951} C_VEL
LIN {X 0,Y 482.616,Z 614.912,A -85,B 0,C 180,E1 -7031.125,E2 -7031.125} C_VEL
LIN {X 0,Y 482.285,Z 622.921,A -85,B 0,C 180,E1 -7032.306,E2 -7032.306} C_VEL
LIN {X 0,Y 482.017,Z 630.399,A -85,B 0,C 180,E1 -7033.706,E2 -7033.706} C_VEL
LIN {X 0,Y 481.757,Z 636.645,A -85,B 0,C 180,E1 -7035.224,E2 -7035.224} C_VEL
LIN {X 0,Y 481.571,Z 640.658,A -85,B 0,C 180,E1 -7036.534,E2 -7036.534} C_VEL
LIN {X 0,Y 481.429,Z 643.557,A -85,B 0,C 180,E1 -7037.853,E2 -7037.853} C_VEL
LIN {X 0,Y 481.405,Z 644.885,A -85,B 0,C 180,E1 -7038.734,E2 -7038.734} C_VEL
LIN {X 0,Y 481.336,Z 645.804,A -85,B 0,C 180,E1 -7039.623,E2 -7039.623} C_VEL
LIN {X 0,Y 481.294,Z 646.305,A -85,B 0,C 180,E1 -7040.849,E2 -7040.849} C_VEL
LIN {X 0,Y 481.298,Z 645.81,A -85,B 0,C 180,E1 -7042.313,E2 -7042.313} C_VEL
LIN {X 0,Y 481.322,Z 644.873,A -85,B 0,C 180,E1 -7043.219,E2 -7043.219} C_VEL
LIN {X 0,Y 481.416,Z 643.462,A -85,B 0,C 180,E1 -7044.127,E2 -7044.127} C_VEL
LIN {X 0,Y 481.541,Z 640.336,A -85,B 0,C 180,E1 -7045.528,E2 -7045.528} C_VEL
LIN {X 0,Y 481.696,Z 636.068,A -85,B 0,C 180,E1 -7046.891,E2 -7046.891} C_VEL
LIN {X 0,Y 481.873,Z 630.235,A -85,B 0,C 180,E1 -7048.295,E2 -7048.295} C_VEL
LIN {X 0,Y 482.173,Z 622.699,A -85,B 0,C 180,E1 -7049.708,E2 -7049.708} C_VEL
LIN {X 0,Y 482.488,Z 614.888,A -85,B 0,C 180,E1 -7050.87,E2 -7050.87} C_VEL
LIN {X 0,Y 482.856,Z 605.798,A -85,B 0,C 180,E1 -7051.968,E2 -7051.968} C_VEL
LIN {X 0,Y 483.122,Z 595.978,A -85,B 0,C 180,E1 -7052.936,E2 -7052.936} C_VEL
LIN {X 0,Y 483.499,Z 585.108,A -85,B 0,C 180,E1 -7053.792,E2 -7053.792} C_VEL
LIN {X 0,Y 483.772,Z 573.403,A -85,B 0,C 180,E1 -7054.512,E2 -7054.512} C_VEL
LIN {X 0,Y 483.989,Z 561.542,A -85,B 0,C 180,E1 -7055.064,E2 -7055.064} C_VEL
LIN {X 0,Y 484.099,Z 548.887,A -85,B 0,C 180,E1 -7055.479,E2 -7055.479} C_VEL
LIN {X 0,Y 484.145,Z 534.618,A -85,B 0,C 180,E1 -7055.752,E2 -7055.752} C_VEL
LIN {X 0,Y 484.039,Z 522.947,A -85,B 0,C 180,E1 -7055.934,E2 -7055.934} C_VEL
LIN {X 0,Y 481.873,Z 516.374,A -85,B 0,C 180,E1 -7056.119,E2 -7056.119} C_VEL
LIN {X 0,Y 481.685,Z 515.396,A -85,B 0,C 180,E1 -7056.281,E2 -7056.281} C_VEL
LIN {X 0,Y 481.676,Z 515.301,A -85,B 0,C 180,E1 -7059.35,E2 -7059.35} C_VEL
LIN {X 0,Y 481.65,Z 515.298,A -85,B 0,C 180,E1 -7062.161,E2 -7062.161} C_VEL
LIN {X 0,Y 481.658,Z 515.301,A -85,B 0,C 180,E1 -7065.544,E2 -7065.544} C_VEL
LIN {X 0,Y 481.671,Z 515.294,A -85,B 0,C 180,E1 -7068.085,E2 -7068.085} C_VEL
LIN {X 0,Y 481.678,Z 515.298,A -85,B 0,C 180,E1 -7069.535,E2 -7069.535} C_VEL
LIN {X 0,Y 481.001,Z 515.379,A -85,B 0,C 180,E1 -7070.232,E2 -7070.232} C_VEL
LIN {X 0,Y 478.119,Z 515.744,A -85,B 0,C 180,E1 -7071.365,E2 -7071.365} C_VEL
LIN {X 0,Y 475.688,Z 516.045,A -85,B 0,C 180,E1 -7072.278,E2 -7072.278} C_VEL
LIN {X 0,Y 474.651,Z 516.172,A -85,B 0,C 180,E1 -7072.984,E2 -7072.984} C_VEL
LIN {X 0,Y 474.57,Z 516.182,A -85,B 0,C 180,E1 -7073.223,E2 -7073.223} C_VEL
LIN {X 0,Y 474.637,Z 516.171,A -85,B 0,C 180,E1 -7076.017,E2 -7076.017} C_VEL
LIN {X 0,Y 474.605,Z 516.178,A -85,B 0,C 180,E1 -7079.191,E2 -7079.191} C_VEL
LIN {X 0,Y 474.699,Z 516.162,A -85,B 0,C 180,E1 -7082.681,E2 -7082.681} C_VEL
LIN {X 0,Y 474.659,Z 516.175,A -85,B 0,C 180,E1 -7085.508,E2 -7085.508} C_VEL
LIN {X 0,Y 474.673,Z 516.168,A -85,B 0,C 180,E1 -7089.186,E2 -7089.186} C_VEL
LIN {X 0,Y 474.649,Z 516.172,A -85,B 0,C 180,E1 -7091.885,E2 -7091.885} C_VEL
LIN {X 0,Y 474.704,Z 516.161,A -85,B 0,C 180,E1 -7094.545,E2 -7094.545} C_VEL
LIN {X 0,Y 474.709,Z 516.164,A -85,B 0,C 180,E1 -7098.038,E2 -7098.038} C_VEL
LIN {X 0,Y 474.731,Z 516.164,A -85,B 0,C 180,E1 -7101.487,E2 -7101.487} C_VEL
LIN {X 0,Y 474.75,Z 516.156,A -85,B 0,C 180,E1 -7104.904,E2 -7104.904} C_VEL
LIN {X 0,Y 474.898,Z 516.142,A -85,B 0,C 180,E1 -7107.456,E2 -7107.456} C_VEL
LIN {X 0,Y 474.917,Z 516.14,A -85,B 0,C 180,E1 -7110,E2 -7110} C_VEL
LIN {X 0,Y 474.899,Z 516.137,A -85,B 0,C 180,E1 -7112.545,E2 -7112.545} C_VEL
LIN {X 0,Y 474.763,Z 516.16,A -85,B 0,C 180,E1 -7115.948,E2 -7115.948} C_VEL
LIN {X 0,Y 474.717,Z 516.16,A -85,B 0,C 180,E1 -7118.514,E2 -7118.514} C_VEL
LIN {X 0,Y 474.709,Z 516.167,A -85,B 0,C 180,E1 -7121.962,E2 -7121.962} C_VEL
LIN {X 0,Y 474.704,Z 516.164,A -85,B 0,C 180,E1 -7125.455,E2 -7125.455} C_VEL
LIN {X 0,Y 474.669,Z 516.166,A -85,B 0,C 180,E1 -7129.01,E2 -7129.01} C_VEL
LIN {X 0,Y 474.592,Z 516.181,A -85,B 0,C 180,E1 -7131.728,E2 -7131.728} C_VEL
LIN {X 0,Y 474.643,Z 516.17,A -85,B 0,C 180,E1 -7134.493,E2 -7134.493} C_VEL
LIN {X 0,Y 474.683,Z 516.165,A -85,B 0,C 180,E1 -7137.334,E2 -7137.334} C_VEL
LIN {X 0,Y 474.607,Z 516.179,A -85,B 0,C 180,E1 -7140.229,E2 -7140.229} C_VEL
LIN {X 0,Y 474.643,Z 516.169,A -85,B 0,C 180,E1 -7143.219,E2 -7143.219} C_VEL
LIN {X 0,Y 474.589,Z 516.18,A -85,B 0,C 180,E1 -7146.323,E2 -7146.323} C_VEL
LIN {X 0,Y 474.65,Z 516.171,A -85,B 0,C 180,E1 -7149.65,E2 -7149.65} C_VEL
LIN {X 0,Y 474.65,Z 516.168,A -85,B 0,C 180,E1 -7152.929,E2 -7152.929} C_VEL
LIN {X 0,Y 474.607,Z 516.179,A -85,B 0,C 180,E1 -7155.894,E2 -7155.894} C_VEL
LIN {X 0,Y 474.625,Z 516.171,A -85,B 0,C 180,E1 -7159.04,E2 -7159.04} C_VEL
LIN {X 0,Y 474.607,Z 516.176,A -85,B 0,C 180,E1 -7161.703,E2 -7161.703} C_VEL
LIN {X 0,Y 474.626,Z 516.173,A -85,B 0,C 180,E1 -7164.725,E2 -7164.725} C_VEL
LIN {X 0,Y 474.633,Z 516.173,A -85,B 0,C 180,E1 -7167.787,E2 -7167.787} C_VEL
LIN {X 0,Y 474.626,Z 516.172,A -85,B 0,C 180,E1 -7170.882,E2 -7170.882} C_VEL
LIN {X 0,Y 474.66,Z 516.168,A -85,B 0,C 180,E1 -7173.628,E2 -7173.628} C_VEL
LIN {X 0,Y 474.629,Z 516.174,A -85,B 0,C 180,E1 -7176.64,E2 -7176.64} C_VEL
LIN {X 0,Y 474.65,Z 516.173,A -85,B 0,C 180,E1 -7180.089,E2 -7180.089} C_VEL
LIN {X 0,Y 474.644,Z 516.172,A -85,B 0,C 180,E1 -7182.774,E2 -7182.774} C_VEL
LIN {X 0,Y 474.64,Z 516.169,A -85,B 0,C 180,E1 -7185.42,E2 -7185.42} C_VEL
LIN {X 0,Y 474.731,Z 516.162,A -85,B 0,C 180,E1 -7188.038,E2 -7188.038} C_VEL
LIN {X 0,Y 474.72,Z 516.159,A -85,B 0,C 180,E1 -7191.486,E2 -7191.486} C_VEL
LIN {X 0,Y 474.78,Z 516.155,A -85,B 0,C 180,E1 -7194.052,E2 -7194.052} C_VEL
LIN {X 0,Y 474.886,Z 516.138,A -85,B 0,C 180,E1 -7197.455,E2 -7197.455} C_VEL
LIN {X 0,Y 474.849,Z 516.147,A -85,B 0,C 180,E1 -7200.848,E2 -7200.848} C_VEL
LIN {X 0,Y 474.886,Z 516.147,A -85,B 0,C 180,E1 -7202.544,E2 -7202.544} C_VEL
LIN {X 0,Y 474.77,Z 516.154,A -85,B 0,C 180,E1 -7205.947,E2 -7205.947} C_VEL
LIN {X 0,Y 474.72,Z 516.168,A -85,B 0,C 180,E1 -7208.513,E2 -7208.513} C_VEL
LIN {X 0,Y 474.694,Z 516.164,A -85,B 0,C 180,E1 -7211.962,E2 -7211.962} C_VEL
LIN {X 0,Y 474.691,Z 516.163,A -85,B 0,C 180,E1 -7215.456,E2 -7215.456} C_VEL
LIN {X 0,Y 474.657,Z 516.171,A -85,B 0,C 180,E1 -7219.01,E2 -7219.01} C_VEL
LIN {X 0,Y 474.581,Z 516.176,A -85,B 0,C 180,E1 -7221.729,E2 -7221.729} C_VEL
LIN {X 0,Y 474.65,Z 516.174,A -85,B 0,C 180,E1 -7224.493,E2 -7224.493} C_VEL
LIN {X 0,Y 474.691,Z 516.164,A -85,B 0,C 180,E1 -7227.339,E2 -7227.339} C_VEL
LIN {X 0,Y 474.603,Z 516.182,A -85,B 0,C 180,E1 -7230.812,E2 -7230.812} C_VEL
LIN {X 0,Y 474.631,Z 516.171,A -85,B 0,C 180,E1 -7233.984,E2 -7233.984} C_VEL
LIN {X 0,Y 474.569,Z 516.185,A -85,B 0,C 180,E1 -7236.9,E2 -7236.9} C_VEL
LIN {X 0,Y 474.621,Z 516.172,A -85,B 0,C 180,E1 -7239.648,E2 -7239.648} C_VEL
LIN {X 0,Y 474.634,Z 516.177,A -85,B 0,C 180,E1 -7242.932,E2 -7242.932} C_VEL
LIN {X 0,Y 474.61,Z 516.173,A -85,B 0,C 180,E1 -7245.896,E2 -7245.896} C_VEL
LIN {X 0,Y 474.627,Z 516.177,A -85,B 0,C 180,E1 -7249.041,E2 -7249.041} C_VEL
LIN {X 0,Y 474.61,Z 516.173,A -85,B 0,C 180,E1 -7251.704,E2 -7251.704} C_VEL
LIN {X 0,Y 474.625,Z 516.179,A -85,B 0,C 180,E1 -7254.727,E2 -7254.727} C_VEL
LIN {X 0,Y 474.634,Z 516.176,A -85,B 0,C 180,E1 -7257.788,E2 -7257.788} C_VEL
LIN {X 0,Y 474.652,Z 516.336,A -85,B 0,C 180,E1 -7259.142,E2 -7259.142} C_VEL
LIN {X 0,Y 477.283,Z 529.207,A -85,B 0,C 180,E1 -7261.649,E2 -7261.649} C_VEL
LIN {X 0,Y 477.395,Z 533.298,A -85,B 0,C 180,E1 -7262.386,E2 -7262.386} C_VEL
LIN {X 0,Y 476.467,Z 553.877,A -85,B 0,C 180,E1 -7265.967,E2 -7265.967} C_VEL
LIN {X 0,Y 475.704,Z 573.086,A -85,B 0,C 180,E1 -7269.233,E2 -7269.233} C_VEL
LIN {X 0,Y 475.163,Z 590.375,A -85,B 0,C 180,E1 -7272.127,E2 -7272.127} C_VEL
LIN {X 0,Y 474.73,Z 610.327,A -85,B 0,C 180,E1 -7275.424,E2 -7275.424} C_VEL
LIN {X 0,Y 474.501,Z 617.757,A -85,B 0,C 180,E1 -7276.607,E2 -7276.607} C_VEL
LIN {X 0,Y 476.212,Z 636.281,A -85,B 0,C 180,E1 -7276.993,E2 -7276.993} C_VEL
LIN {X 0,Y 476.455,Z 646.127,A -85,B 0,C 180,E1 -7277.164,E2 -7277.164} C_VEL
LIN {X 0,Y 476.062,Z 698.94,A -85,B 0,C 180,E1 -7278.05,E2 -7278.05} C_VEL
LIN {X 0,Y 475.711,Z 710.085,A -85,B 0,C 180,E1 -7278.388,E2 -7278.388} C_VEL
LIN {X 0,Y 475.395,Z 721.602,A -85,B 0,C 180,E1 -7278.92,E2 -7278.92} C_VEL
LIN {X 0,Y 475.014,Z 731.816,A -85,B 0,C 180,E1 -7279.558,E2 -7279.558} C_VEL
LIN {X 0,Y 474.622,Z 742.243,A -85,B 0,C 180,E1 -7280.411,E2 -7280.411} C_VEL
LIN {X 0,Y 474.409,Z 750.501,A -85,B 0,C 180,E1 -7281.266,E2 -7281.266} C_VEL
LIN {X 0,Y 474.199,Z 758.765,A -85,B 0,C 180,E1 -7282.335,E2 -7282.335} C_VEL
LIN {X 0,Y 474.129,Z 764.667,A -85,B 0,C 180,E1 -7283.283,E2 -7283.283} C_VEL
LIN {X 0,Y 474.014,Z 770.547,A -85,B 0,C 180,E1 -7284.47,E2 -7284.47} C_VEL
LIN {X 0,Y 474.009,Z 775.369,A -85,B 0,C 180,E1 -7285.749,E2 -7285.749} C_VEL
LIN {X 0,Y 474.017,Z 777.76,A -85,B 0,C 180,E1 -7286.6,E2 -7286.6} C_VEL
LIN {X 0,Y 473.976,Z 779.584,A -85,B 0,C 180,E1 -7287.45,E2 -7287.45} C_VEL
LIN {X 0,Y 473.954,Z 780.855,A -85,B 0,C 180,E1 -7288.301,E2 -7288.301} C_VEL
LIN {X 0,Y 473.951,Z 781.591,A -85,B 0,C 180,E1 -7289.15,E2 -7289.15} C_VEL
LIN {X 0,Y 474.071,Z 781.847,A -85,B 0,C 180,E1 -7290,E2 -7290} C_VEL
LIN {X 0,Y 473.961,Z 781.513,A -85,B 0,C 180,E1 -7290.85,E2 -7290.85} C_VEL
LIN {X 0,Y 473.974,Z 780.703,A -85,B 0,C 180,E1 -7291.699,E2 -7291.699} C_VEL
LIN {X 0,Y 474.005,Z 779.335,A -85,B 0,C 180,E1 -7292.549,E2 -7292.549} C_VEL
LIN {X 0,Y 474.06,Z 776.276,A -85,B 0,C 180,E1 -7293.825,E2 -7293.825} C_VEL
LIN {X 0,Y 474.02,Z 771.8,A -85,B 0,C 180,E1 -7295.103,E2 -7295.103} C_VEL
LIN {X 0,Y 474.117,Z 766.795,A -85,B 0,C 180,E1 -7296.196,E2 -7296.196} C_VEL
LIN {X 0,Y 474.131,Z 760.769,A -85,B 0,C 180,E1 -7297.238,E2 -7297.238} C_VEL
LIN {X 0,Y 474.316,Z 753.053,A -85,B 0,C 180,E1 -7298.306,E2 -7298.306} C_VEL
LIN {X 0,Y 474.589,Z 744.375,A -85,B 0,C 180,E1 -7299.267,E2 -7299.267} C_VEL
LIN {X 0,Y 474.839,Z 734.646,A -85,B 0,C 180,E1 -7300.123,E2 -7300.123} C_VEL
LIN {X 0,Y 475.191,Z 723.637,A -85,B 0,C 180,E1 -7300.869,E2 -7300.869} C_VEL
LIN {X 0,Y 475.486,Z 713.238,A -85,B 0,C 180,E1 -7301.402,E2 -7301.402} C_VEL
LIN {X 0,Y 475.906,Z 700.415,A -85,B 0,C 180,E1 -7301.85,E2 -7301.85} C_VEL
LIN {X 0,Y 476.054,Z 687.903,A -85,B 0,C 180,E1 -7302.102,E2 -7302.102} C_VEL
LIN {X 0,Y 476.267,Z 637.654,A -85,B 0,C 180,E1 -7302.91,E2 -7302.91} C_VEL
LIN {X 0,Y 474.537,Z 614.988,A -85,B 0,C 180,E1 -7303.352,E2 -7303.352} C_VEL
LIN {X 0,Y 474.531,Z 612.314,A -85,B 0,C 180,E1 -7303.707,E2 -7303.707} C_VEL
LIN {X 0,Y 474.832,Z 591.724,A -85,B 0,C 180,E1 -7306.996,E2 -7306.996} C_VEL
LIN {X 0,Y 475.291,Z 571.151,A -85,B 0,C 180,E1 -7310.333,E2 -7310.333} C_VEL
LIN {X 0,Y 475.774,Z 552.025,A -85,B 0,C 180,E1 -7313.505,E2 -7313.505} C_VEL
LIN {X 0,Y 476.4,Z 533.09,A -85,B 0,C 180,E1 -7316.739,E2 -7316.739} C_VEL
LIN {X 0,Y 476.544,Z 526.404,A -85,B 0,C 180,E1 -7317.917,E2 -7317.917} C_VEL
LIN {X 0,Y 474.68,Z 516.333,A -85,B 0,C 180,E1 -7319.856,E2 -7319.856} C_VEL
LIN {X 0,Y 474.639,Z 516.176,A -85,B 0,C 180,E1 -7323.219,E2 -7323.219} C_VEL
LIN {X 0,Y 474.588,Z 516.18,A -85,B 0,C 180,E1 -7326.323,E2 -7326.323} C_VEL
